// TwinCAT 3 PLC project LabController
// ProgramVersion: 3.1.4022.1
// libraries:
//   Tc2_MC2, * (Beckhoff Automation GmbH)
//   Tc2_Standard, * (Beckhoff Automation GmbH)
//   Tc2_System, * (Beckhoff Automation GmbH)
//   Tc2_Utilities, * (Beckhoff Automation GmbH)
//   Tc3_Module, * (Beckhoff Automation GmbH)
// project tree:
//   DUTs/Control/ ST_Control.TcDUT, ST_ControlComau.TcDUT, ST_ControlStewart.TcDUT, ST_ControlWinch.TcDUT
//   DUTs/ E_MotionLabState.TcDUT
//   DUTs/Feedback/ ST_Feedback.TcDUT, ST_FeedbackComau.TcDUT, ST_FeedbackLeica.TcDUT, ST_FeedbackMru.TcDUT, ST_FeedbackQualisys.TcDUT, ST_FeedbackStewart.TcDUT, ST_FeedbackWinch.TcDUT
//   DUTs/QualisysRT/Components/ ST_3DMarkerPositionNoLabel.TcDUT, ST_3DMarkerPositionNoLabelComponent.TcDUT, ST_RT6D.TcDUT, ST_RT6DComponent.TcDUT
//   DUTs/QualisysRT/ E_ComponentType.TcDUT, ST_RTComponentData.TcDUT, ST_RTDataQRTPacket.TcDUT
//   DUTs/RxHmi/ ST_RxHmi.TcDUT
//   DUTs/RxUdp/ ST_RxUdpComau.TcDUT, ST_RxUdpMru.TcDUT, ST_RxUdpQualisys.TcDUT, ST_RxUdpRemote.TcDUT, ST_RxUdpStewart.TcDUT
//   DUTs/TxHmi/ ST_TxHmi.TcDUT, ST_TxHmiComau.TcDUT, ST_TxHmiMru.TcDUT, ST_TxHmiQualisys.TcDUT, ST_TxHmiStewart.TcDUT, ST_TxHmiWinch.TcDUT
//   DUTs/TxUdp/ ST_TxUdpComau.TcDUT, ST_TxUdpRemote.TcDUT, ST_TxUdpStewart.TcDUT
//   / GVL.TcGVL, MainTask.TcTTO
//   HydroSimulator/ E_TcMatSimDataAreaType.TcDUT, FB_HydroSimulator.TcPOU, FB_TcMatSimObject.TcPOU, ST_HydroSimulatorInitData.TcDUT, ST_HydroSimulator_Input.TcDUT, ST_HydroSimulator_Output.TcDUT, ST_TcMatSimObjectDataAreaInfo.TcDUT
//   POUs/CSV/ FB_CsvReader.TcPOU
//   POUs/Interfaces/ E_ComauMode.TcDUT, E_StewartCommand.TcDUT, E_StewartMode.TcDUT, E_StewartOpMode.TcDUT, E_StewartState.TcDUT, E_StewartStatus.TcDUT, E_WinchMode.TcDUT, FB_ComauInterface.TcPOU, FB_LeicaInterface.TcPOU, FB_MruInterface.TcPOU, FB_QualisysInterface.TcPOU, FB_RemoteInterface.TcPOU, FB_WinchInterface.TcPOU, FB_StewartInterface.TcPOU
//   POUs/ MAIN.TcPOU
//   POUs/Simulink/ FB_QuatToRotMatrix.TcPOU
//   POUs/UdpFBs/ FB_UdpServerRT.TcPOU, FB_UdpClientRT.TcPOU
//   POUs/Utils/ FB_SoftMotion.TcPOU, F_VelocityBoundary.TcPOU, ST_VelocityBoundary.TcDUT
//   SystemFunctions/ CheckDivReal.TcPOU, CheckDivLReal.TcPOU
// real-time tasks:
//   TASK SimTask: cycle T#5ms, priority 21, ADS port 351
//   TASK MainTask: cycle T#5ms, priority 20, ADS port 350
// motion (NC):
//   TASK NC-Task 1 SAF: cycle T#1ms, priority 4, ADS port 501
//   TASK NC-Task 1 SVB: cycle T#5ms, priority 8, ADS port 511
//   AXIS RobotWinch (id 1) // Winch placed on top of Comau Robot
//     General: UnitName=m
//     Dynamic: AccelerationMaximum=10000, DecelerationMaximum=10000, Acceleration=3.56741726765625, Deceleration=3.56741726765625, Jerk=10.7022518029688
//     Velo: RefSearch=0.023782781784375, RefSync=0.023782781784375, SlowManual=0.118913908921875, FastManual=0.71348345353125, Fast=2.3782781784375, Maximum=2.3782781784375
//     OtherSettings: AllowMotionCmdToSlave=true
//     encoder EncType=8
//       EncPara: ScaleFactorNumerator=0.0218304, ScaleFactorDenominator=1048576, Inverse=true, MaxCount=#xffffffff
//         SoftEndMinControl: Enable=true, Range=-7.5
//         SoftEndMaxControl: Enable=true, Range=-6
//     drive DrvType=9
//       DrvPara: Inverse=true, MaxCount=#xffffffff, DriveControlDWord=#x00030100
//         Analog: VeloReferenz=2.61610599628125, VeloScale=1.02400649589962, ScaleFactorActTorque=0.1
//         TimeComp: TaskDelayCycles=1
//     controller CtrType=1
//       CtrPara: PriorControlFactor=1
//         PosDiffControl: Enable=false, Range=10
//         Observer: BandWidth=20
// I/O:
//   DEVICE EM8000 (RT-Ethernet Adapter)
//   DEVICE EM1500 (RT-Ethernet Adapter)
//   DEVICE MRU1 (RT-Ethernet Adapter)
//   DEVICE MRU2 (RT-Ethernet Adapter)
//   DEVICE COMAU (RT-Ethernet Adapter)
//   DEVICE EtherCAT, AmsNetId 169.254.76.98.11.1
//     Drive 1 (AX5103-0000-0210) [AX5103-0000-0210 EtherCAT Drive (SoE, 1 Ch.)]
//     Box 1 (Leica-RT-Output) [Leica RT Output] (disabled)
//   DEVICE REMOTE (RT-Ethernet Adapter)
//   DEVICE QTM (RT-Ethernet Adapter)
// variable links:
//   NC-Task 1 SAF/Axes/RobotWinch <-> EtherCAT/Drive 1 (AX5103-0000-0210)
//     Drive/Inputs/In/nDataIn1 <-> AT/Following distance
//     Drive/Inputs/In/nDcOutputTime <-> InfoData/DcOutputShift
//     Drive/Inputs/In/nState1 <-> AT/Drive status word @bit 8
//     Drive/Inputs/In/nState2 <-> AT/Drive status word
//     Drive/Inputs/In/nState4 @bit 1 <-> WcState/InputToggle
//     Drive/Inputs/In/nState4 <-> WcState/WcState
//     Drive/Outputs/Out/nCtrl1 <-> MDT/Master control word @bit 8
//     Drive/Outputs/Out/nDataOut1 <-> MDT/Position command value
//     Enc/Inputs/In/nDataIn1 <-> AT/Position feedback 1 value
//     Enc/Inputs/In/nDcInputTime <-> InfoData/DcInputShift
//     Enc/Inputs/In/nState4 @bit 1 <-> WcState/InputToggle
//     Enc/Inputs/In/nState4 <-> WcState/WcState
//   LabController/LabController Instance <-> NC-Task 1 SAF/Axes/RobotWinch
//     MainTask Inputs/MAIN.winch.axis.NcToPlc <-> Outputs/ToPlc
//     MainTask Outputs/MAIN.winch.axis.PlcToNc <-> Inputs/FromPlc

CONFIGURATION LabController
    RESOURCE PLC ON TwinCAT3
        TASK MainTask(INTERVAL := T#5ms, PRIORITY := 20);
        PROGRAM MAIN WITH MainTask : MAIN;
    END_RESOURCE
END_CONFIGURATION

// ---- DUTs/Control/ST_Control.TcDUT
TYPE ST_Control :
STRUCT
	em8000: ST_ControlStewart;
	em1500: ST_ControlStewart;
	comau: ST_ControlComau;
	winch: ST_ControlWinch;
END_STRUCT
END_TYPE

// ---- DUTs/Control/ST_ControlComau.TcDUT
TYPE ST_ControlComau :
STRUCT
	u : ARRAY[0..5] OF LREAL;

END_STRUCT
END_TYPE

// ---- DUTs/Control/ST_ControlStewart.TcDUT
TYPE ST_ControlStewart :
STRUCT
	// Velocity setpint to stewart
	u : ARRAY[0..5] OF LREAL;
	
END_STRUCT
END_TYPE

// ---- DUTs/Control/ST_ControlWinch.TcDUT
TYPE ST_ControlWinch :
STRUCT
	length : LREAL;
	length_t : LREAL;
	length_tt : LREAL;
END_STRUCT
END_TYPE

// ---- DUTs/E_MotionLabState.TcDUT
{attribute 'qualified_only'}
{attribute 'strict'}
TYPE E_MotionLabState :
(
	STOP := 16#00,
	NORMAL := 16#01,
	ERROR := 16#10
) USINT;
END_TYPE

// ---- DUTs/Feedback/ST_Feedback.TcDUT
TYPE ST_Feedback :
STRUCT
	em8000: ST_FeedbackStewart;
	em1500: ST_FeedbackStewart;
	mru1: ST_FeedbackMru;
	mru2: ST_FeedbackMru;
	comau: ST_FeedbackComau;
	winch: ST_FeedbackWinch;
	qtm: ST_FeedbackQualisys;
	at960: ST_FeedbackLeica;
END_STRUCT
END_TYPE

// ---- DUTs/Feedback/ST_FeedbackComau.TcDUT
TYPE ST_FeedbackComau :
STRUCT
	q: ARRAY[0..5] OF LREAL;
	q_t: ARRAY[0..5] OF LREAL;
END_STRUCT
END_TYPE

// ---- DUTs/Feedback/ST_FeedbackLeica.TcDUT
TYPE ST_FeedbackLeica :
STRUCT
	pos: ARRAY[0..2] OF LREAL;
	R11: LREAL;
	R12: LREAL;
	R13: LREAL;
	R21: LREAL;
	R22: LREAL;
	R23: LREAL;
	R31: LREAL;
	R32: LREAL;
	R33: LREAL;
END_STRUCT
END_TYPE

// ---- DUTs/Feedback/ST_FeedbackMru.TcDUT
TYPE ST_FeedbackMru :
STRUCT
	eta: ARRAY[0..5] OF LREAL;
	v: ARRAY[0..5] OF LREAL;
END_STRUCT
END_TYPE

// ---- DUTs/Feedback/ST_FeedbackQualisys.TcDUT
TYPE ST_FeedbackQualisys :
STRUCT
	dist: LREAL;
	pos: ARRAY[0..2] OF LREAL;
END_STRUCT
END_TYPE

// ---- DUTs/Feedback/ST_FeedbackStewart.TcDUT
TYPE ST_FeedbackStewart :
STRUCT
	eta: ARRAY[0..5] OF LREAL;
	eta_t: ARRAY[0..5] OF LREAL;
	eta_tt: ARRAY[0..5] OF LREAL;
END_STRUCT
END_TYPE

// ---- DUTs/Feedback/ST_FeedbackWinch.TcDUT
TYPE ST_FeedbackWinch :
STRUCT
	length: LREAL;
	length_t: LREAL;
END_STRUCT
END_TYPE

// ---- DUTs/QualisysRT/Components/ST_3DMarkerPositionNoLabel.TcDUT
TYPE ST_3DMarkerPositionNoLabel :
STRUCT
	x : REAL;
	y : REAL;
	z : REAL;
	id : DINT;
END_STRUCT
END_TYPE

// ---- DUTs/QualisysRT/Components/ST_3DMarkerPositionNoLabelComponent.TcDUT
TYPE ST_3DMarkerPositionNoLabelComponent :
STRUCT
	nSize : UDINT;
	nType : UDINT;
	nMarkers : UDINT;
	nDropRate : INT;
	nOutOfSyncRate : INT;
	markers : ARRAY [0..99] OF ST_3DMarkerPositionNoLabel;
END_STRUCT
END_TYPE

// ---- DUTs/QualisysRT/Components/ST_RT6D.TcDUT
TYPE ST_RT6D :
STRUCT
	x : REAL;
	y : REAL;
	z : REAL;
	rotMatrix : ARRAY [0..8] OF REAL;
END_STRUCT
END_TYPE

// ---- DUTs/QualisysRT/Components/ST_RT6DComponent.TcDUT
TYPE ST_RT6DComponent :
STRUCT
	nSize : UDINT;
	nType : UDINT;
	nBodies : UDINT;
	nDropRate : INT;
	nOutOfSyncRate : INT;
	bodies : ARRAY [0..99] OF ST_RT6D;
END_STRUCT
END_TYPE

// ---- DUTs/QualisysRT/E_ComponentType.TcDUT
{attribute 'qualified_only'}
{attribute 'strict'}
TYPE E_ComponentType :
(
	e3D := 1, // 3D marker data
	e3DNoLabel := 2, //Unidentified 3D marker data
	eAnalog := 3, // Analog data from available analog devices
	eForce := 4, // Force data from available force plates.
	e6D := 5, // 6D data - position and rotation matrix
	e6DEuler := 6, // 6D data - position and Euler angles
	e2D := 7, // 2D marker data
	e2DLinearized := 8, // Linearized 2D marker data
	e3DResiduals := 9, // 3D marker data with residuals
 	e3DNoLabelsResiduals := 10, // Unidentified 3D marker data with residuals
	e6DResiduals := 11, // 6D data - position and rotation matrix with residuals
	e6DEulerResiduals := 12, // 6D data - position and Euler angles with residuals
	eAnalogSingle := 13, // Analog data from available analog devices. Only one sample per channel and camera frame. The latest sample is used if more than one sample is available.
	eImage := 14, // Image frame from a specific camera. Image size and format is set with the XML settings, see Image settings.
	eForceSingle := 15 // Force data from available force plates. Only one sample per plate and camera frame. The latest sample is used if more than one sample is available.
);
END_TYPE

// ---- DUTs/QualisysRT/ST_RTComponentData.TcDUT
TYPE ST_RTComponentData :
STRUCT
	nSize : UDINT;
	nType : UDINT;
END_STRUCT
END_TYPE

// ---- DUTs/QualisysRT/ST_RTDataQRTPacket.TcDUT
TYPE ST_RTDataQRTPacket :
STRUCT
	nSize : UDINT;
	nType : UDINT;
	nTimestamp : LINT;
	nFramenumber : UDINT;
	nComponentCount : UDINT;
END_STRUCT
END_TYPE

// ---- DUTs/RxHmi/ST_RxHmi.TcDUT
TYPE ST_RxHmi :
STRUCT
	counter : UDINT := 0;
	winchJogUp : BOOL;
	winchJogDown : BOOL;
	xboxLeftX : REAL;
	xboxLeftY : REAL;
	xboxRightX : REAL;
	xboxRightY : REAL;
	xboxLT : REAL;
	xboxRT : REAL;
END_STRUCT
END_TYPE

// ---- DUTs/RxUdp/ST_RxUdpComau.TcDUT
TYPE ST_RxUdpComau :
STRUCT
	frameCounter : DINT := 0;
	q 		: ARRAY [0..5] OF REAL;
	q_t 	: ARRAY [0..5] OF REAL;
	qMin 	: ARRAY [0..5] OF REAL;
	qMax 	: ARRAY [0..5] OF REAL;
	qMax_t 	: ARRAY [0..5] OF REAL;
END_STRUCT
END_TYPE

// ---- DUTs/RxUdp/ST_RxUdpMru.TcDUT
{attribute 'pack_mode' := '1'}
TYPE ST_RxUdpMru :
STRUCT
	mruOK : BYTE; // Mru Status, 113=OK
	dataLength : BYTE; // Data length
	token : BYTE; // MRU token
	SystemTime : DINT; // No. 176 - [ms] - Sample time in milliseconds since power on
	SensorTemp : REAL; // No. 31 - [DegC] - Sensor house temprature     
	AngRate_D : REAL; // No. 9 - [rad/s] - Angular rate in Down direction (h-frame). Turn Rate
	Roll : REAL; // No. 63 - [rad] - Roll angle (euler angle)
	Pitch : REAL; // No. 64 - [rad] - Pitch angle (euler angle)
	Yaw : REAL; // No. 65 - [rad] - Yaw angle (euler angle)
	AngRate_R : REAL; // No. 1 - [rad/s] - Angular rate in roll axis (b-frame)
	AngRate_P : REAL; // No. 2 - [rad/s] - Angular rate in pitch axis (b-frame)
	AngRate_Y : REAL; // No. 3 - [rad/s] - Angular rate in yaw axis (b-frame)
	VelMru_R : REAL; // No. 244 - [m/s] - Linear velocity at MRU point in R-direction (b-frame)
	VelMru_P : REAL; // No. 245 - [m/s] - Linear velocity at MRU point in P-direction (b-frame)
	VelMru_Y : REAL; // No. 246 - [m/s] - Linear velocity at MRU point in Y-direction (b-frame)
	AccMru_R : REAL; // No. 238 - [m/s] - Linear acceleration at MRU point in R-direction (b-frame)
	AccMru_P : REAL; // No. 239 - [m/s] - Linear acceleration at MRU point in P-direction (b-frame)
	AccMru_Y : REAL; // No. 240 - [m/s] - Linear acceleration at MRU point in Y-direction (b-frame)
	PosCg_F : REAL; // No. 274 - [m] - Linear position at CG in forward direction (h-frame)
	PosCg_S : REAL; // No. 275 - [m] - Linear position at CG in starboard direction (h-frame)
	PosCg_D : REAL; // No. 276 - [m] - Linear position at CG in down direction (h-frame)
	VelCg_F : REAL; // No. 262 - [m/s] - Linear velocity at CG in forward direction (h-frame)
	VelCg_S : REAL; // No. 263 - [m/s] - Linear velocity at CG in starboard direction (h-frame)
	VelCg_D : REAL; // No. 264 - [m/s] - Linear velocity at CG in down direction (h-frame)
	AccCg_F : REAL; // No. 250 - [m/s2] - Linear acceleration (raw/unfiltered) at CG in forward direction (h-frame)
	AccCg_S : REAL; // No. 251 - [m/s2] - Linear acceleration (raw/unfiltered) at CG in starboard direction (h-frame)
	AccCg_D : REAL; // No. 252 - [m/s2] - Linear acceleration (raw/unfiltered) at CG in down direction (h-frame)
	checksum : BYTE; // Data checksum 
END_STRUCT
END_TYPE

// ---- DUTs/RxUdp/ST_RxUdpQualisys.TcDUT
TYPE ST_RxUdpQualisys :
STRUCT
	// Header
	dataSize : UDINT;
	dataType : UDINT;
	timestamp : ULINT;
	frameNumber : UDINT;
	componentCount : UDINT;
	// Component
	componentSize : UDINT;
	componentType : UDINT;
END_STRUCT
END_TYPE

// ---- DUTs/RxUdp/ST_RxUdpRemote.TcDUT
TYPE ST_RxUdpRemote :
STRUCT
	iUdpKey : UDINT; // Udp Key
	iCounter : UDINT; // Heartbeat counter
	eModeCmd : UDINT; // Operation mode
	em8000_u : ARRAY [0..5] OF REAL; // EM8000 DOF position setpoints
	em8000_u_t : ARRAY [0..5] OF REAL; // EM8000 DOF velocity setpoints
	em1500_u : ARRAY [0..5] OF REAL; // EM1500 DOF position setpoints
	em1500_u_t : ARRAY [0..5] OF REAL; // EM1500 DOF velocity setpoints
	comau_u : ARRAY [0..5] OF REAL; // Joint speed setpoints
	winch_u : REAL; // Winch wire speed setpoint
	
END_STRUCT
END_TYPE

// ---- DUTs/RxUdp/ST_RxUdpStewart.TcDUT
TYPE ST_RxUdpStewart :
STRUCT
	Frame_Count : UDINT := 0;
	Motion_Status : UDINT := 0;
	Platform_setpoint_surge : REAL := 0.0;
	Platform_setpoint_sway : REAL := 0.0;
	Platform_setpoint_heave : REAL := 0.0;
	Platform_setpoint_roll : REAL := 0.0;
	Platform_setpoint_pitch : REAL := 0.0;
	Platform_setpoint_yaw : REAL := 0.0;
	Special_effect_surge_setpoint : REAL := 0.0;
	Special_effect_sway_setpoint : REAL := 0.0;
	Special_effect_heave_setpoint : REAL := 0.0;
	Special_effect_roll_setpoint : REAL := 0.0;
	Special_effect_pitch_setpoint : REAL := 0.0;
	Special_effect_yaw_setpoint : REAL := 0.0;
	Actual_position_actuator_1 : REAL := 0.0;
	Actual_position_actuator_2 : REAL := 0.0;
	Actual_position_actuator_3 : REAL := 0.0;
	Actual_position_actuator_4 : REAL := 0.0;
	Actual_position_actuator_5 : REAL := 0.0;
	Actual_position_actuator_6 : REAL := 0.0;
	Actual_platform_position_surge : REAL := 0.0;
	Actual_platform_position_sway : REAL := 0.0;
	Actual_platform_position_heave : REAL := 0.0;
	Actual_platform_position_roll : REAL := 0.0;
	Actual_platform_position_pitch : REAL := 0.0;
	Actual_platform_position_yaw : REAL := 0.0;
	Actual_platform_velocity_surge : REAL := 0.0;
	Actual_platform_velocity_sway : REAL := 0.0;
	Actual_platform_velocity_heave : REAL := 0.0;
	Actual_platform_velocity_roll : REAL := 0.0;
	Actual_platform_velocity_pitch : REAL := 0.0;
	Actual_platform_velocity_yaw : REAL := 0.0;
	Actual_platform_acceleration_surge : REAL := 0.0;
	Actual_platform_acceleration_sway : REAL := 0.0;
	Actual_platform_acceleration_heave : REAL := 0.0;
	Actual_platform_acceleration_roll : REAL := 0.0;
	Actual_platform_acceleration_pitch : REAL := 0.0;
	Actual_platform_acceleration_yaw : REAL := 0.0;
END_STRUCT
END_TYPE

// ---- DUTs/TxHmi/ST_TxHmi.TcDUT
TYPE ST_TxHmi :
STRUCT
	em8000 : ST_TxHmiStewart;
	em1500 : ST_TxHmiStewart;
	mru1 : ST_TxHmiMru;
	mru2 : ST_TxHmiMru;
	comau : ST_TxHmiComau;
	winch : ST_TxHmiWinch;
	qtm : ST_TxHmiQualisys;
	phi : ARRAY [0..1] OF REAL;
	phi_t : ARRAY [0..1] OF REAL;	
	e : ARRAY [0..2] OF REAL;
	c : REAL;
END_STRUCT
END_TYPE

// ---- DUTs/TxHmi/ST_TxHmiComau.TcDUT
TYPE ST_TxHmiComau :
STRUCT
	status : DINT;
	u : ARRAY [0..5] OF REAL;
	q : ARRAY [0..5] OF REAL;
	q_t : ARRAY [0..5] OF REAL;
	qMin : ARRAY [0..5] OF REAL;
	qMax : ARRAY [0..5] OF REAL;
	qMax_t : ARRAY [0..5] OF REAL;
END_STRUCT
END_TYPE

// ---- DUTs/TxHmi/ST_TxHmiMru.TcDUT
TYPE ST_TxHmiMru :
STRUCT
	status : DINT := 0;
	eta : ARRAY [0..5] OF REAL;
END_STRUCT
END_TYPE

// ---- DUTs/TxHmi/ST_TxHmiQualisys.TcDUT
TYPE ST_TxHmiQualisys :
STRUCT
	status : DINT;
	dist : REAL;
	x : REAL;
	y : REAL;
	z : REAL;
	markers : ARRAY [0..9] OF ST_3DMarkerPositionNoLabel;
END_STRUCT
END_TYPE

// ---- DUTs/TxHmi/ST_TxHmiStewart.TcDUT
TYPE ST_TxHmiStewart :
STRUCT
	status : DINT := 0;
	eta : ARRAY [0..5] OF REAL;
	etaRef : ARRAY [0..5] OF REAL;
	cyl : ARRAY [0..5] OF REAL;
	dofScale : ARRAY [0..5] OF REAL;
END_STRUCT
END_TYPE

// ---- DUTs/TxHmi/ST_TxHmiWinch.TcDUT
TYPE ST_TxHmiWinch :
STRUCT
	status : DINT := 0;
	l : REAL;
END_STRUCT
END_TYPE

// ---- DUTs/TxUdp/ST_TxUdpComau.TcDUT
TYPE ST_TxUdpComau :
STRUCT
	udpKey : DINT := 0;
	cmnd : DINT; // 0: SETTLED, 1: ENGAGED
	qDotRef : ARRAY [0..5] OF REAL;
END_STRUCT
END_TYPE

// ---- DUTs/TxUdp/ST_TxUdpRemote.TcDUT
TYPE ST_TxUdpRemote :
STRUCT
	// Mode and time
	eMode : UDINT;
	t : REAL;
	
	// Equipement: Comau robot
	comau_q : ARRAY [0..5] OF REAL;
	comau_q_t : ARRAY [0..5] OF REAL;
	
	// Equipement: Robot Winch
	winch_l : REAL;
	winch_l_t : REAL;

	// Equipement: EM8000
	em8000_eta : ARRAY [0..5] OF REAL;
	em8000_eta_t : ARRAY [0..5] OF REAL;
	em8000_eta_tt : ARRAY [0..5] OF REAL;
	
	// Equipement: MRU1 (Mounted on EM8000)
	mru1_eta : ARRAY [0..5] OF REAL;
	mru1_v : ARRAY [0..5] OF REAL;
	
	// Equipement: EM1500 and MRU2
	em1500_eta : ARRAY [0..5] OF REAL;
	em1500_eta_t : ARRAY [0..5] OF REAL;
	em1500_eta_tt : ARRAY [0..5] OF REAL;
	
	// Equipement: MRU2 (Mounted on EM1500)
	mru2_eta : ARRAY [0..5] OF REAL;
	mru2_v : ARRAY [0..5] OF REAL;
	
END_STRUCT
END_TYPE

// ---- DUTs/TxUdp/ST_TxUdpStewart.TcDUT
TYPE ST_TxUdpStewart :
STRUCT
	COUNT : UDINT := 0;
	CMND : UDINT := 0;
	AX : REAL := 0.0;
	AY : REAL := 0.0;
	AZ : REAL := 0.0;
	Dax : REAL := 0.0;
	Day : REAL := 0.0;
	Daz : REAL := 0.0;
	P_dot_CG : REAL := 0.0;
	Q_dot_CG : REAL := 0.0;
	R_dot_CG : REAL := 0.0;
	P_CG : REAL := 0.0;
	Q_CG : REAL := 0.0;
	R_CG : REAL := 0.0;
	Phi : REAL := 0.0;
	Theta : REAL := 0.0;
	U : REAL := 0.0;
	X_DIRECT : REAL := 0.0;
	Y_DIRECT : REAL := 0.0;
	Z_DIRECT : REAL := 0.0;
	X_CG : REAL := 0.0;
	Y_CG : REAL := 0.0;
	Z_CG : REAL := 0.0;
	Flags : REAL := 0.0;
	Bump_1 : REAL := 0.0;
	Bump_2 : REAL := 0.0;
	Bump_3 : REAL := 0.0;
	Bump_4 : REAL := 0.0;
	Bump_5 : REAL := 0.0;
	FREQ1 : REAL := 0.0;
	FREQ2 : REAL := 0.0;
	FREQ3 : REAL := 0.0;
	FREQ4 : REAL := 0.0;
	FREQ5 : REAL := 0.0;
	FREQ6 : REAL := 0.0;
	FREQ7 : REAL := 0.0;
	FREQ8 : REAL := 0.0;
	FREQ9 : REAL := 0.0;
	FREQ10 : REAL := 0.0;
	FREQ11 : REAL := 0.0;
	FREQ12 : REAL := 0.0;
	FREQ13 : REAL := 0.0;
	FREQ14 : REAL := 0.0;
	FREQ15 : REAL := 0.0;
	FREQ16 : REAL := 0.0;
	FREQ17 : REAL := 0.0;
	FREQ18 : REAL := 0.0;
	FREQ19 : REAL := 0.0;
	FREQ20 : REAL := 0.0;
	XGAIN1 : REAL := 0.0;
	XGAIN2 : REAL := 0.0;
	XGAIN3 : REAL := 0.0;
	XGAIN4 : REAL := 0.0;
	XGAIN5 : REAL := 0.0;
	XGAIN6 : REAL := 0.0;
	XGAIN7 : REAL := 0.0;
	XGAIN8 : REAL := 0.0;
	XGAIN9 : REAL := 0.0;
	XGAIN10 : REAL := 0.0;
	XGAIN11 : REAL := 0.0;
	XGAIN12 : REAL := 0.0;
	XGAIN13 : REAL := 0.0;
	XGAIN14 : REAL := 0.0;
	XGAIN15 : REAL := 0.0;
	XGAIN16 : REAL := 0.0;
	XGAIN17 : REAL := 0.0;
	XGAIN18 : REAL := 0.0;
	XGAIN19 : REAL := 0.0;
	XGAIN20 : REAL := 0.0;
	YGAIN1 : REAL := 0.0;
	YGAIN2 : REAL := 0.0;
	YGAIN3 : REAL := 0.0;
	YGAIN4 : REAL := 0.0;
	YGAIN5 : REAL := 0.0;
	YGAIN6 : REAL := 0.0;
	YGAIN7 : REAL := 0.0;
	YGAIN8 : REAL := 0.0;
	YGAIN9 : REAL := 0.0;
	YGAIN10 : REAL := 0.0;
	YGAIN11 : REAL := 0.0;
	YGAIN12 : REAL := 0.0;
	YGAIN13 : REAL := 0.0;
	YGAIN14 : REAL := 0.0;
	YGAIN15 : REAL := 0.0;
	YGAIN16 : REAL := 0.0;
	YGAIN17 : REAL := 0.0;
	YGAIN18 : REAL := 0.0;
	YGAIN19 : REAL := 0.0;
	YGAIN20 : REAL := 0.0;
	ZGAIN1 : REAL := 0.0;
	ZGAIN2 : REAL := 0.0;
	ZGAIN3 : REAL := 0.0;
	ZGAIN4 : REAL := 0.0;
	ZGAIN5 : REAL := 0.0;
	ZGAIN6 : REAL := 0.0;
	ZGAIN7 : REAL := 0.0;
	ZGAIN8 : REAL := 0.0;
	ZGAIN9 : REAL := 0.0;
	ZGAIN10 : REAL := 0.0;
	ZGAIN11 : REAL := 0.0;
	ZGAIN12 : REAL := 0.0;
	ZGAIN13 : REAL := 0.0;
	ZGAIN14 : REAL := 0.0;
	ZGAIN15 : REAL := 0.0;
	ZGAIN16 : REAL := 0.0;
	ZGAIN17 : REAL := 0.0;
	ZGAIN18 : REAL := 0.0;
	ZGAIN19 : REAL := 0.0;
	ZGAIN20 : REAL := 0.0;
	X_EXTRA : REAL := 0.0;
	Y_EXTRA : REAL := 0.0;
	Z_EXTRA : REAL := 0.0;
	PHI_EXTRA : REAL := 0.0;
	THETA_EXTRA : REAL := 0.0;
	PSI_EXTRA : REAL := 0.0;
	X_EXTRA_DOT : REAL := 0.0;
	Y_EXTRA_DOT : REAL := 0.0;
	Z_EXTRA_DOT : REAL := 0.0;
	PHI_EXTRA_DOT : REAL := 0.0;
	THETA_EXTRA_DOT : REAL := 0.0;
	PSI_EXTRA_DOT : REAL := 0.0;
	X_EXTRA_DDOT : REAL := 0.0;
	Y_EXTRA_DDOT : REAL := 0.0;
	Z_EXTRA_DDOT : REAL := 0.0;
	PHI_EXTRA_DDOT : REAL := 0.0;
	THETA_EXTRA_DDOT : REAL := 0.0;
	PSI_EXTRA_DDOT : REAL := 0.0;
END_STRUCT
END_TYPE

// ---- HydroSimulator/E_TcMatSimDataAreaType.TcDUT
TYPE E_TcMatSimDataAreaType :
(
	NotSpecified := 0,
	Standard,
	InputSrc,
	InputDst,
	OutputSrc,
	OutputDst,
	InternalDa,
	MArea,
	RetainDa
);
END_TYPE

// ---- HydroSimulator/ST_HydroSimulatorInitData.TcDUT
{attribute 'pack_mode' := '4'}
TYPE ST_HydroSimulatorInitData :
STRUCT
	Header: TComInitDataHdr;
	CallByHdr: TComInitDataElmHdr;
	CallBy: TctModuleCallByType;
	ExecutionSequenceHdr: TComInitDataElmHdr;
	ExecutionSequence: TctModuleExecutionSequenceType;
	StepSizeHdr: TComInitDataElmHdr;
	StepSize: TctStepSizeType;
	ExecuteModelCodeHdr: TComInitDataElmHdr;
	ExecuteModelCode: BOOL;
	ModelParametersHdr: TComInitDataElmHdr;
	ModelParameters: P_HydroSimulator_T;
	ContextInfoArr_0_TaskOidHdr: TComInitDataElmHdr;
	ContextInfoArr_0_TaskOid: OTCID;
	ContextInfoArr_0_TaskPriorityHdr: TComInitDataElmHdr;
	ContextInfoArr_0_TaskPriority: UDINT;
	ContextInfoArr_0_TaskCycleTimeNsHdr: TComInitDataElmHdr;
	ContextInfoArr_0_TaskCycleTimeNs: UDINT;
	ContextInfoArr_0_TaskPortHdr: TComInitDataElmHdr;
	ContextInfoArr_0_TaskPort: UINT;
	ContextInfoArr_0_TaskSortOrderHdr: TComInitDataElmHdr;
	ContextInfoArr_0_TaskSortOrder: UDINT;
END_STRUCT
END_TYPE

// ---- HydroSimulator/ST_HydroSimulator_Input.TcDUT
TYPE ST_HydroSimulator_Input :
STRUCT
	bReset: BOOL;
	etaMax: matrix_6_real_T := [0.1, 0.1, 0.3, 5.0/180.0*PI, 5.0/180.0*PI, 5.0/180.0*PI];
	w0 : LREAL := 0.5457;
	lambda : LREAL := 0.2405;
	sigma : LREAL := 0.8444;
	
END_STRUCT
END_TYPE

// ---- HydroSimulator/ST_HydroSimulator_Output.TcDUT
TYPE ST_HydroSimulator_Output :
STRUCT
	scale: matrix_6_real_T;
	eta: matrix_6_real_T;
	v: matrix_6_real_T;
	v_t: matrix_6_real_T;
END_STRUCT
END_TYPE

// ---- HydroSimulator/ST_TcMatSimObjectDataAreaInfo.TcDUT
TYPE ST_TcMatSimObjectDataAreaInfo :
STRUCT
	pPlcVar: PVOID;
	pModuleProcImg: PVOID;
	nSize: UDINT;
	nDataAreaId: UDINT;
	eDataAreaType: E_TcMatSimDataAreaType;
END_STRUCT
END_TYPE

// ---- POUs/Interfaces/E_ComauMode.TcDUT
{attribute 'qualified_only'}
{attribute 'strict'}
TYPE E_ComauMode :
(
	SETTLED := 0,
	REMOTE,
	MOTION_COMP
) DINT;
END_TYPE

// ---- POUs/Interfaces/E_StewartCommand.TcDUT
{attribute 'qualified_only'}
{attribute 'strict'}
TYPE E_StewartCommand :
(
	TO_OFF	 		:= 16#00000000,
	TO_SETTLED 		:= 16#00000001,
	TO_NEUTRAL 		:= 16#00000003,
	TO_ENGAGED 		:= 16#00000007,
	ACK_FAULT 		:= 16#00000011 // Akcnowledge fault and go to settled
) UDINT;
END_TYPE

// ---- POUs/Interfaces/E_StewartMode.TcDUT
{attribute 'qualified_only'}
{attribute 'strict'}
TYPE E_StewartMode :
(
	SETTLED := 0,
	NEUTRAL,
	SIMULATION,
	GENERATOR,
	REMOTE
) USINT ;
END_TYPE

// ---- POUs/Interfaces/E_StewartOpMode.TcDUT
{attribute 'qualified_only'}
{attribute 'strict'}
TYPE E_StewartOpMode :
(
	MANUAL 	:= 16#00,
	NORMAL	:= 16#01
) USINT;
END_TYPE

// ---- POUs/Interfaces/E_StewartState.TcDUT
{attribute 'qualified_only'}
{attribute 'strict'}
TYPE E_StewartState :
(
	TRANSIT 		:= 16#00,
	OFF				:= 16#01,
	SETTLED			:= 16#02,
	OIL_HEATING		:= 16#03,
	NEUTRAL 		:= 16#04,
	NEUTRAL_FREEZE	:= 16#05,
	ENGAGED			:= 16#08,
	ENGAGED_FREEZE	:= 16#09	
) USINT;
END_TYPE

// ---- POUs/Interfaces/E_StewartStatus.TcDUT
{attribute 'qualified_only'}
{attribute 'strict'}
TYPE E_StewartStatus :
(
	SYSTEM_OK 	:= 16#00,
	WARNING		:= 16#04,
	ERROR		:= 16#08
) USINT;
END_TYPE

// ---- POUs/Interfaces/E_WinchMode.TcDUT
{attribute 'qualified_only'}
{attribute 'strict'}
TYPE E_WinchMode :
(
	SETTLED := 0,
	LOCAL,
	REMOTE,
	MOTION_COMP
) USINT;
END_TYPE

// ---- POUs/Utils/ST_VelocityBoundary.TcDUT
TYPE ST_VelocityBoundary :
STRUCT
	qMin_t : LREAL;
	qMax_t : LREAL;
END_STRUCT
END_TYPE

// ---- GVL.TcGVL
{attribute 'qualified_only'}
VAR_GLOBAL
	logMessage : STRING(255) := 'No Message';
END_VAR

// ---- POUs/MAIN.TcPOU
PROGRAM MAIN
VAR_INPUT
	bStop : BOOL;
	bReset : BOOL := FALSE;
	
END_VAR
VAR_OUTPUT
	eState : E_MotionLabState;
	
END_VAR
VAR
	// TEST/DEBUG
	rand : DRAND;
	k : UINT;
	data : ARRAY [0..9] OF REAL;

	// Task monitoring
	fbGetCurrentTaskIdx : GETCURTASKINDEX;
	bCycleTimeExceeded : BOOL;
	nCycleCount : UDINT;
	Ts : LREAL;
	t : LREAL;
	
	// Linear wave parameters, Hs = 8 and Tp = 12.0;
	w0 AT %Q* : LREAL := 0.5457;
	lambda AT %Q* : LREAL := 0.2405;
	sigma AT %Q* : LREAL := 1.5012;
	
	// HMI data
	txHmi : ST_TxHmi;
	rxHmi : ST_RxHmi;
	
	// HMI activity check
	hmiCounterOld : UDINT := 0;
	hmiTimer : TON;
	
	// Remote interface
	remote : FB_RemoteInterface('192.168.90.60', 50060, 50050); // CPU-X001
	
	// Machinery
	em8000 : FB_StewartInterface('192.168.90.30', 50030, 50040, oid:=16#01010060);
	em1500 : FB_StewartInterface('192.168.90.31', 50031, 50041, oid:=16#01010070);
	comau : FB_ComauInterface('192.168.90.32', 50032, 50042);
	winch : FB_WinchInterface(ADR(txHmi.winch));
	
	// Sensors
	mru1 : FB_MruInterface(50043, ADR(txHmi.mru1));
	mru2 : FB_MruInterface(50044, ADR(txHmi.mru2));
	qtm : FB_QualisysInterface(50199, ADR(txHmi.qtm));
	at960 : FB_LeicaInterface;
	
	// Hydro simulators
	
	
	
	// System call for starting PqQt HMI
	fbStartProcess : NT_StartProcess;
	
	phi : ARRAY [0..1] OF LREAL;
END_VAR

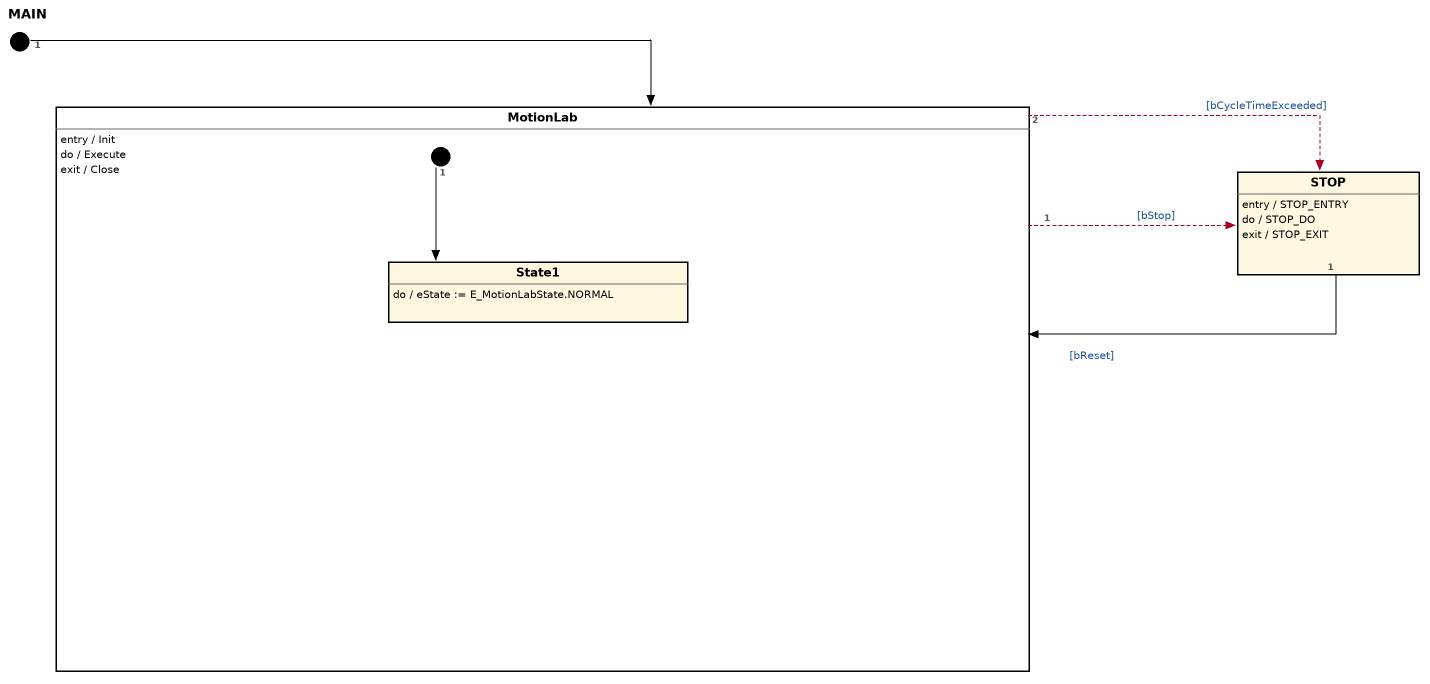
STATECHART MAIN  // abortable
    START StartState1
    COMPOSITE STATE MotionLab
        entry / Init
        do / Execute
        exit / Close
        START StartState2
        STATE State1
            do / eState := E_MotionLabState.NORMAL
        StartState2 -> State1  // priority 1, on completion
    END_STATE
    STATE STOP
        entry / STOP_ENTRY
        do / STOP_DO
        exit / STOP_EXIT
    StartState1 -> MotionLab  // priority 1, on completion
    MotionLab -> STOP [bStop] // priority 1, exception
    MotionLab -> STOP [bCycleTimeExceeded] // priority 2, exception
    STOP -> MotionLab [bReset] // priority 1
END_STATECHART

METHOD Close : BOOL
VAR_INPUT
END_VAR
END_METHOD

METHOD PRIVATE Execute : BOOL
VAR_INPUT
END_VAR
VAR
	i : UINT;

END_VAR
// Task monitoring
fbGetCurrentTaskIdx();
bCycleTimeExceeded := _TaskInfo[fbGetCurrentTaskIdx.index].CycleTimeExceeded;
nCycleCount := _TaskInfo[fbGetCurrentTaskIdx.index].CycleCount;
Ts := UDINT_TO_LREAL(_TaskInfo[fbGetCurrentTaskIdx.index].CycleTime/10)/1E6;


FOR i := 0 TO 9 DO
	data[i] := LREAL_TO_REAL((1 + i)*0.1*SIN(0.1*2*PI*t));
END_FOR

// Update all interfaces
em8000(
	Ts := Ts,
);
em1500(
	Ts := Ts,
);

mru1();
mru2();
at960();
qtm();
comau();

winch(
	Ts := Ts
);


// *** REMOTE Interface ***
// PLC -> REMOTE
remote.feedback.em8000 := em8000.feedback;
remote.feedback.mru1 := mru1.feedback;

remote.feedback.em1500 := em1500.feedback;
remote.feedback.mru2 := mru2.feedback;

remote.feedback.comau.q := comau.q;

// Execute remote
remote(
	Ts := Ts
);

// REMOTE -> PLC
em1500.bRemoteActive := remote.bActive;
em1500.uRemote := remote.control.em1500.u;
em1500.uRemote_t := remote.control.em1500.u_t;

// *** REMOTE Interface ***
END_METHOD

METHOD Init : BOOL
VAR_INPUT
END_VAR
END_METHOD

METHOD PRIVATE STOP_DO : BOOL
VAR_INPUT
END_VAR

// Update all interfaces
Execute();

eState := E_MotionLabState.STOP;
END_METHOD

METHOD PRIVATE STOP_ENTRY : BOOL
VAR_INPUT
END_VAR
em8000.bStop := TRUE;
em1500.bStop := TRUE;
END_METHOD

METHOD PRIVATE STOP_EXIT : BOOL
VAR_INPUT
END_VAR
bStop := FALSE;
bReset := FALSE;

// Reset equipement
em8000.bReset := TRUE;
em1500.bReset := TRUE;
END_METHOD

END_PROGRAM

// ---- POUs/Interfaces/FB_RemoteInterface.TcPOU
FUNCTION_BLOCK FB_RemoteInterface
VAR_INPUT
	Ts : LREAL := 0.005;
	// feedback from motion lab
	feedback : ST_Feedback;
	
	
END_VAR
VAR_OUTPUT
	// Activity status
	bActive : BOOL := FALSE;
	
	// Control to motion lab
	control : ST_Control;
	
END_VAR
VAR
	// Udp connection
	rxUdp : ST_RxUdpRemote;
	txUdp : ST_TxUdpRemote;
	udpClient : FB_UdpClientRT('', 0, 0, 0, 0, 0, 0);	// Dummy constructor
	
	// Timer
	iCounterOld : UDINT := 0;
	fbTimer : TON;
	
	
	i : UINT;
	
END_VAR

// Feedback data
FOR i := 0 TO 5 DO
	// eMode
	txUdp.eMode := 0;
	
	// Time 
	txUdp.t := txUdp.t + LREAL_TO_REAL(Ts);
	
	// EM8000
	txUdp.em8000_eta[i] := LREAL_TO_REAL(feedback.em8000.eta[i]);
	txUdp.em8000_eta_t[i] := LREAL_TO_REAL(feedback.em8000.eta_t[i]);
	txUdp.em8000_eta_tt[i] := LREAL_TO_REAL(feedback.em8000.eta_tt[i]);
	
	// MRU1
	txUdp.mru1_eta[i] := LREAL_TO_REAL(feedback.mru1.eta[i]);
	txUdp.mru1_v[i] := LREAL_TO_REAL(feedback.mru1.v[i]);
	
	// EM1500
	txUdp.em1500_eta[i] := LREAL_TO_REAL(feedback.em1500.eta[i]);
	txUdp.em1500_eta_t[i] := LREAL_TO_REAL(feedback.em1500.eta_t[i]);
	txUdp.em1500_eta_tt[i] := LREAL_TO_REAL(feedback.em1500.eta_tt[i]);
	
	// MRU1
	txUdp.mru2_eta[i] := LREAL_TO_REAL(feedback.mru2.eta[i]);
	txUdp.mru2_v[i] := LREAL_TO_REAL(feedback.mru2.v[i]);
	
	
	// COMAU
	
	
	
END_FOR

// WINCH



// Update Udp client
udpClient();

// Control data
FOR i := 0 TO 5 DO
	// EM8000
	control.em8000.u[i] := REAL_TO_LREAL(rxUdp.em8000_u[i]);
	
	// MRU1
	
	
	// EM1500
	control.em1500.u[i] := REAL_TO_LREAL(rxUdp.em1500_u[i]);
	
	// MRU2
	
	// COMAU
	
	
END_FOR

// WINCH




// Timeout setting
fbTimer.PT := T#500MS;

IF rxUdp.iCounter <> iCounterOld THEN
	// Update old counter
	iCounterOld := rxUdp.iCounter;
	
	// Reset timeout timer
	fbTimer(
		IN := FALSE
	);
	
ELSE
	// Start timout timer
	fbTimer(
		IN := TRUE
	);
	
END_IF

// Set bActive based on timer
bActive := NOT fbTimer.Q;

METHOD FB_exit : BOOL
VAR_INPUT
	bInCopyCode : BOOL; // if TRUE, the exit method is called for exiting an instance that is copied afterwards (online change).
END_VAR
END_METHOD

METHOD FB_init : BOOL
VAR_INPUT
	bInitRetains : BOOL; // if TRUE, the retain variables are initialized (warm start / cold start)
	bInCopyCode : BOOL;  // if TRUE, the instance afterwards gets moved into the copy code (online change)
	
	// Init variables
	_remoteIpAddr : T_Ipv4Addr;
	_remotePort : UINT;
	_localPort : UINT;
END_VAR
// Initilize udpClient
udpClient.FB_init(
	bInitRetains,
	bInCopyCode,
	_remoteIpAddr,
	_remotePort,
	_localPort,
	SIZEOF(rxUdp),
	ADR(rxUdp),
	SIZEOF(txUdp),
	ADR(txUdp)
);
END_METHOD

METHOD FB_reinit : BOOL
VAR_INPUT
END_VAR
END_METHOD

END_FUNCTION_BLOCK

// ---- POUs/UdpFBs/FB_UdpClientRT.TcPOU
{attribute 'c++_compatible'}
FUNCTION_BLOCK FB_UdpClientRT IMPLEMENTS ITcIoUdpProtocolRecv
VAR_INPUT
	
END_VAR
VAR_OUTPUT
END_VAR
VAR
	// ITcIoUdpProtocolRecv related 
	{attribute 'TcInitSymbol'}
	oid : OTCID; 
	ipUdp : ITcIoUdpProtocol;
	
	// Initilized variables
	remoteIpAddr : UDINT;
	remotePort : UINT;
	localPort : UINT;
	{attribute 'tc_no_symbol'}
	nRxData : UDINT := 0;
	{attribute 'tc_no_symbol'}
	pRxData : PVOID;
	{attribute 'tc_no_symbol'}
	nTxData : UDINT := 0;
	{attribute 'tc_no_symbol'}
	pTxData : PVOID;
	
	// Send/Recv counters
	rxCounter : UINT;
	txCounter : UINT;
	
	// Result
	hrInit : HRESULT;
	hrSend : HRESULT;
END_VAR

IF ipUdp <> 0 THEN
	// Send data to remote server
	IF nTxData > 0 THEN		
		hrSend := ipUdp.SendData(remoteIpAddr, remotePort, localPort, nTxData, pTxData, TRUE, 0);
		txCounter := txCounter + 1;
	END_IF
	
	// Check for incoming data
	IF nRxData > 0 THEN
		ipUdp.CheckReceived();
	END_IF
END_IF

{attribute 'conditionalshow'}
METHOD FB_exit : BOOL
VAR_INPUT
	bInCopyCode : BOOL; // if TRUE, the exit method is called for exiting an instance that is copied afterwards (online change).
END_VAR
IF NOT bInCopyCode THEN // no online change
	IF ipUdp <> 0 THEN 
		ipUdp.UnregisterReceiver(localPort); // Shutdown
		FW_SafeRelease(ADR(ipUdp));
		FB_exit := TRUE; 
	END_IF
END_IF
END_METHOD

{attribute 'conditionalshow'}
METHOD FB_init : BOOL
VAR_INPUT
	bInitRetains : BOOL; // if TRUE, the retain variables are initialized (warm start / cold start)
	bInCopyCode : BOOL;  // if TRUE, the instance afterwards gets moved into the copy code (online change)
	
	// Init variables
	_remoteIpAddr : T_Ipv4Addr;
	_remotePort : UINT;
	_localPort : UINT;
	_nRxData : UDINT;
	_pRxData : PVOID;
	_nTxData : UDINT;
	_pTxData : PVOID;
END_VAR
VAR
    ipSrv : ITComObjectServer;
	ipArr : T_IPv4AddrArr;
	i : UINT;
END_VAR
// Initilize member variables
remoteIpAddr := IpToLong(_remoteIpAddr);
remotePort := _remotePort;
localPort := _localPort;
nRxData := _nRxData;
pRxData := _pRxData;
nTxData := _nTxData;
pTxData := _pTxData;

IF NOT bInCopyCode THEN // no online change
	IF ipUdp = 0 THEN
	    hrInit := FW_ObjMgr_GetObjectInstance(
			oid:=oid, 
			iid:=TC_GLOBAL_IID_LIST.IID_ITcIoUdpProtocol, 
			pipUnk:=ADR(ipUdp)
		);
		
		IF SUCCEEDED(hrInit) THEN 
			IF  SUCCEEDED(ipUdp.RegisterReceiver(localPort, THIS^)) THEN //open port
				FB_init := TRUE;
			ELSE 
				FW_SafeRelease(ADR(ipUdp));
			END_IF
		END_IF				
	END_IF
END_IF
END_METHOD

{attribute 'conditionalshow'}
METHOD FB_reinit : BOOL
VAR_INPUT
END_VAR
IF (ipUdp <> 0) THEN 
	ipUdp.RegisterReceiver(localPort, THIS^);
	FB_reinit := TRUE; 
END_IF
END_METHOD

METHOD IpToLong : UDINT
VAR_INPUT
	ipAddr : T_Ipv4Addr;
END_VAR

VAR
	ipAddrArr : T_Ipv4AddrArr;
	ipAddrLong : UDINT;
END_VAR
// Scan ip string to byte array
ipAddrArr := F_ScanIPv4AddrIds(ipAddr);

// Copy bytes to ipaddrLong in reverse direction
MEMCPY(ADR(ipAddrLong) + 0, ADR(ipAddrArr) + 3, 1);
MEMCPY(ADR(ipAddrLong) + 1, ADR(ipAddrArr) + 2, 1);
MEMCPY(ADR(ipAddrLong) + 2, ADR(ipAddrArr) + 1, 1);
MEMCPY(ADR(ipAddrLong) + 3, ADR(ipAddrArr) + 0, 1); 

// Return long ip adress
IpToLong := ipAddrLong;
END_METHOD

{attribute 'object_name' := 'ReceiveData'}
{attribute 'c++_compatible'}
{attribute 'signature_flag' := '33554688'}
{attribute 'pack_mode' := '4'}
{attribute 'show'}
{attribute 'minimal_input_size' := '4'}
METHOD ReceiveData : HRESULT
VAR_INPUT
	ipAddr	: UDINT;
	udpDestPort	: UINT;
	udpSrcPort	: UINT;
	nData	: UDINT;
	pData	: PVOID;
	pVlan	: POINTER TO ETYPE_VLAN_HEADER := 0;
END_VAR
// Check data size and copy data
IF nData = nRxData THEN
	// Copy recived data
	MEMCPY(pRxData, pData, nRxData);
	
	// Increment counters
	rxCounter := rxCounter + 1;
END_IF
END_METHOD

{attribute 'object_name' := 'TcAddRef'}
{attribute 'c++_compatible'}
{attribute 'signature_flag' := '33554688'}
{attribute 'pack_mode' := '4'}
{attribute 'show'}
{attribute 'minimal_input_size' := '4'}
METHOD TcAddRef : UDINT
END_METHOD

{attribute 'object_name' := 'TcQueryInterface'}
{attribute 'c++_compatible'}
{attribute 'signature_flag' := '33554688'}
{attribute 'pack_mode' := '4'}
{attribute 'show'}
{attribute 'minimal_input_size' := '4'}
METHOD TcQueryInterface : HRESULT
VAR_INPUT
	iid	: REFERENCE TO IID;
	pipItf	: POINTER TO PVOID;
END_VAR
VAR
	ipUdpRecv : ITcIoUdpProtocolRecv;
	ipUnknown : ITcUnknown;	
END_VAR
IF GuidsEqual(ADR(iid), ADR(TC_GLOBAL_IID_LIST.IID_ITcIoUdpProtocolRecv)) THEN
	ipUdpRecv := THIS^; // cast to interface pointer
	pipItf^ := ITCUNKNOWN_TO_PVOID(ipUdpRecv);
	TcAddRef();
	TcQueryInterface := S_OK;
ELSIF GuidsEqual(ADR(iid), ADR(TC_GLOBAL_IID_LIST.IID_ITcUnknown)) THEN
	ipUnknown := THIS^; // cast to interface pointer
	pipItf^ := ITCUNKNOWN_TO_PVOID(ipUnknown);
	TcAddRef();
	TcQueryInterface := S_OK;
ELSE
	TcQueryInterface := E_HRESULTAdsErr.NOINTERFACE ; //Call super if this fb extends some other
END_IF
END_METHOD

{attribute 'object_name' := 'TcRelease'}
{attribute 'c++_compatible'}
{attribute 'signature_flag' := '33554688'}
{attribute 'pack_mode' := '4'}
{attribute 'show'}
{attribute 'minimal_input_size' := '4'}
METHOD TcRelease : UDINT
END_METHOD

END_FUNCTION_BLOCK

// ---- POUs/Interfaces/FB_StewartInterface.TcPOU
FUNCTION_BLOCK FB_StewartInterface
VAR_INPUT
	// PLC task time step
	Ts : LREAL := 0.005;
	
	// Stewart Operation 
	bStop : BOOL;
	bReset : BOOL;
	bResetScale : BOOL;
	bStart : BOOL;
	eModeCmd : E_StewartMode;
	
	// Remote data input
	bRemoteActive : BOOL := FALSE;
	uRemote : ARRAY [0..5] OF LREAL;
	uRemote_t : ARRAY [0..5] OF LREAL;
	
END_VAR
VAR_OUTPUT
	bError : BOOL;
	bBusy : BOOL := FALSE;
	bReady : BOOL := FALSE;
	eState : E_StewartState;
	eStatus : E_StewartStatus;
	eOpMode : E_StewartOpMode;
	eMode : E_StewartMode;
	
	// Feedback data
	feedback : ST_FeedbackStewart;
	
	(*
	eta : ARRAY [0..5] OF LREAL;
	eta_t : ARRAY [0..5] OF LREAL;
	eta_tt : ARRAY [0..5] OF LREAL;
	*)
	
END_VAR
VAR	
	// Hydro Simualator
	hydro : FB_HydroSimulator(0);
	
	// Stewart positon input
	u : ARRAY [0..5] OF LREAL;
	u_t : ARRAY [0..5] OF LREAL;
	uOld : ARRAY [0..5] OF LREAL;
	
	// Limted stewart setpoints
	etaRef : ARRAY [0..5] OF LREAL;
	etaRef_t : ARRAY [0..5] OF LREAL;
	etaRef_tt : ARRAY [0..5] OF LREAL;
	etaRefOld : ARRAY [0..5] OF LREAL;

	// Sine wave data
	etaSine : ARRAY [0..5] OF LREAL;
	etaSine_t : ARRAY [0..5] OF LREAL;
	etaSine_tt : ARRAY [0..5] OF LREAL;
	
	// Udp connection
	udpClient : FB_UdpClientRT('', 0, 0, 0, 0, 0, 0);	// Dummy constructor

	{attribute 'tc_no_symbol'}
	eCmnd : E_StewartCommand;
	{attribute 'tc_no_symbol'}
	rxUdp : ST_RxUdpStewart;
	{attribute 'tc_no_symbol'}
	txUdp : ST_TxUdpStewart;
	
	// Hmi connection
	txHmi : ST_TxHmiStewart;
	
	// Udp activity monitoring
	bActive : BOOL;
	frame : UDINT := 0;
	frameOld : UDINT := 0;
	frameLoss : UDINT := 0;
	
	// Time
	t : LREAL := 0.0;
	
	// Sine Generator Settings
	sineAmplitude : ARRAY [0..5] OF LREAL := [0, 0, 0.2, 2.0/180.0*PI, 2.0/180.0*PI, 0];
	sineOmega : ARRAY [0..5] OF LREAL := [0.6283, 0.6283, 0.6283, 0.6283, 0.6283, 0.6283];
	sinePhase : ARRAY [0..5] OF LREAL;

	// Zero eta
	{attribute 'tc_no_symbol'}
	etaZeros : ARRAY [0..5] OF LREAL;
	
	// Max/min settings
	etaRefMin : ARRAY [0..5] OF LREAL;
	etaRefMax : ARRAY [0..5] OF LREAL;
	
	// Soft Motion Input for Remote
	fbSoftMotion : ARRAY [0..5] OF FB_SoftMotion;
	
END_VAR

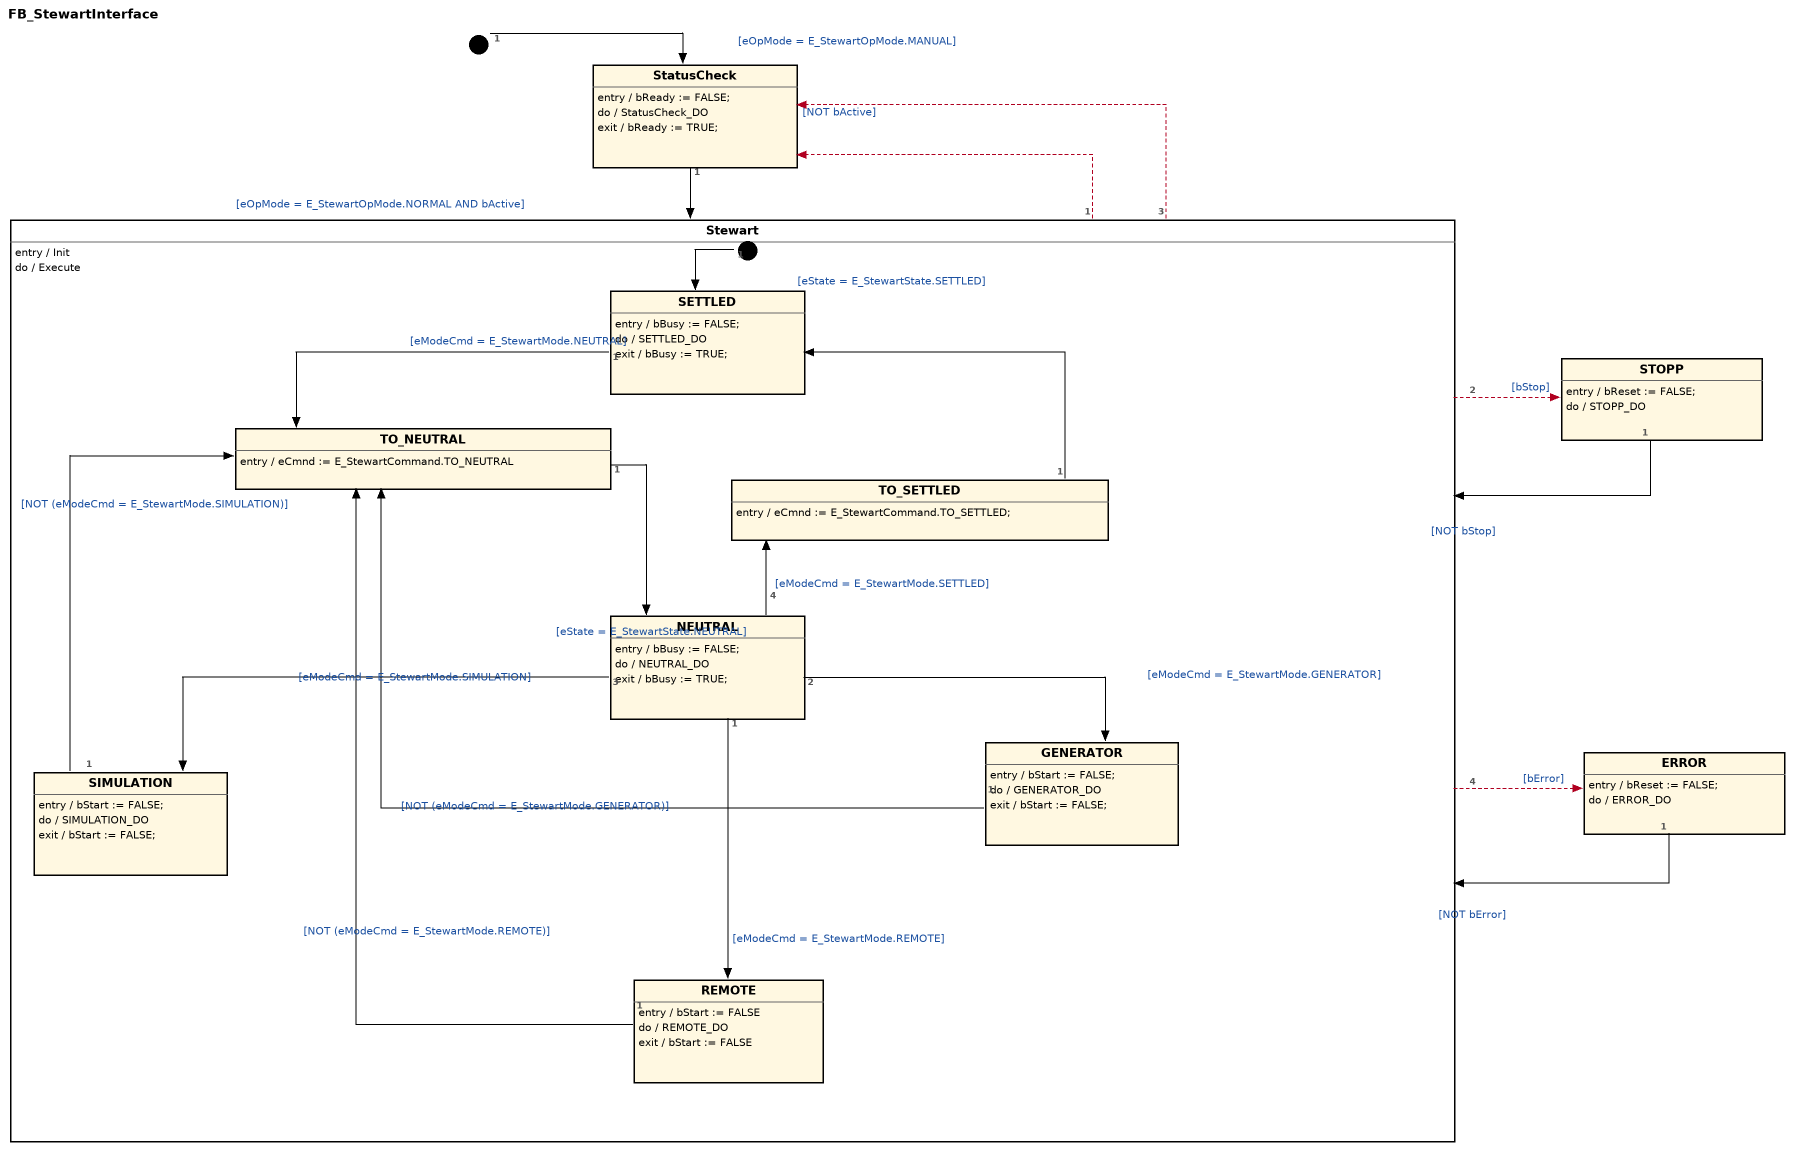
STATECHART ST_StewartInterface  // abortable
    START StartState1
    STATE StatusCheck
        entry / bReady := FALSE;
        do / StatusCheck_DO
        exit / bReady := TRUE;
    COMPOSITE STATE Stewart
        entry / Init
        do / Execute
        START StartState2
        STATE SETTLED
            entry / bBusy := FALSE;
            do / SETTLED_DO
            exit / bBusy := TRUE;
        STATE TO_NEUTRAL
            entry / eCmnd := E_StewartCommand.TO_NEUTRAL
        STATE TO_SETTLED
            entry / eCmnd := E_StewartCommand.TO_SETTLED;
        STATE NEUTRAL
            entry / bBusy := FALSE;
            do / NEUTRAL_DO
            exit / bBusy := TRUE;
        STATE GENERATOR
            entry / bStart := FALSE;
            do / GENERATOR_DO
            exit / bStart := FALSE;
        STATE SIMULATION
            entry / bStart := FALSE;
            do / SIMULATION_DO
            exit / bStart := FALSE;
        STATE REMOTE
            entry / bStart := FALSE
            do / REMOTE_DO
            exit / bStart := FALSE
        StartState2 -> SETTLED  // priority 1, on completion
        SETTLED -> TO_NEUTRAL [eModeCmd = E_StewartMode.NEUTRAL] // priority 1
        TO_NEUTRAL -> NEUTRAL [eState = E_StewartState.NEUTRAL] // priority 1
        TO_SETTLED -> SETTLED [eState = E_StewartState.SETTLED] // priority 1
        NEUTRAL -> REMOTE [eModeCmd = E_StewartMode.REMOTE] // priority 1
        NEUTRAL -> GENERATOR [eModeCmd = E_StewartMode.GENERATOR] // priority 2
        NEUTRAL -> SIMULATION [eModeCmd = E_StewartMode.SIMULATION] // priority 3
        NEUTRAL -> TO_SETTLED [eModeCmd = E_StewartMode.SETTLED] // priority 4
        GENERATOR -> TO_NEUTRAL [NOT (eModeCmd = E_StewartMode.GENERATOR)] // priority 1
        SIMULATION -> TO_NEUTRAL [NOT (eModeCmd = E_StewartMode.SIMULATION)] // priority 1
        REMOTE -> TO_NEUTRAL [NOT (eModeCmd = E_StewartMode.REMOTE)] // priority 1
    END_STATE
    STATE STOPP
        entry / bReset := FALSE;
        do / STOPP_DO
    STATE ERROR
        entry / bReset := FALSE;
        do / ERROR_DO
    StartState1 -> StatusCheck  // priority 1, on completion
    StatusCheck -> Stewart [eOpMode = E_StewartOpMode.NORMAL AND bActive] // priority 1
    Stewart -> StatusCheck [NOT bActive] // priority 1, exception
    Stewart -> STOPP [bStop] // priority 2, exception
    Stewart -> StatusCheck [eOpMode = E_StewartOpMode.MANUAL] // priority 3, exception
    Stewart -> ERROR [bError] // priority 4, exception
    STOPP -> Stewart [NOT bStop] // priority 1
    ERROR -> Stewart [NOT bError] // priority 1
END_STATECHART

METHOD decode_E_StewartOpMode : E_StewartOpMode
VAR_INPUT
	motionStatus : UDINT;
END_VAR
VAR
	mask : UDINT;
	n : USINT;
END_VAR

mask := 16#FF000000 AND motionStatus;
n := UDINT_TO_USINT(SHR(mask, 6));

(*
CASE mask OF
	16#00000000 :
		eResult := E_StewartOpMode.MANUAL;
		
	16#01000000 :
		eResult := E_StewartOpMode.NORMAL;
	
END_CASE
*)
END_METHOD

METHOD PRIVATE decode_E_StewartState : E_StewartState
VAR_INPUT
	motionStatus : UDINT;
END_VAR
VAR
	mask : UDINT;
	eResult : E_StewartState;
END_VAR
// PDF: Motion System Ethernet Interface p.18

mask := 16#0000000F AND motionStatus;

CASE mask OF
	16#00000000 : 
		eResult := E_StewartState.TRANSIT;
		
	16#00000001 : 
		eResult := E_StewartState.OFF;
		
	16#00000002 : 
		eResult := E_StewartState.SETTLED;
		
	16#00000003 : 
		eResult := E_StewartState.OIL_HEATING;
		
	16#00000004 : 
		eResult := E_StewartState.NEUTRAL;
		
	16#00000005 : 
		eResult := E_StewartState.NEUTRAL_FREEZE;
		
	16#00000008 : 
		eResult := E_StewartState.ENGAGED;
		
	16#00000009 : 
		eResult := E_StewartState.ENGAGED_FREEZE;
	
END_CASE

decode_E_StewartState := eResult;
END_METHOD

METHOD decode_E_StewartStatus : E_StewartStatus
VAR_INPUT
	motionStatus : UDINT;
END_VAR
VAR
	mask : UDINT;
	eResult : E_StewartStatus;
END_VAR

mask := 16#000000F0 AND motionStatus;

CASE mask OF
	16#00000000 :
		eResult := E_StewartStatus.SYSTEM_OK;
		
	16#01000040 :
		eResult := E_StewartStatus.WARNING;
		
	16#01000080 :
		eResult := E_StewartStatus.ERROR;
	
END_CASE

decode_E_StewartStatus := eResult;
END_METHOD

METHOD PRIVATE ERROR_DO : BOOL
VAR_INPUT
END_VAR
// Wait for SYSTEM_OK and return to settled
IF eStatus = E_StewartStatus.SYSTEM_OK THEN
	eModeCmd := E_StewartMode.SETTLED;
	eCmnd := E_StewartCommand.TO_SETTLED;

	bError := FALSE;
	
END_IF

// Check for bReset request and acknowledge fault
IF bReset THEN
	eCmnd := E_StewartCommand.ACK_FAULT;
	bReset := FALSE;
END_IF

// Execute main thread
Execute();
END_METHOD

METHOD PRIVATE Execute : BOOL
VAR_INPUT
END_VAR
VAR

	i: INT;
	
	nState : DWORD;
	nStatus : DWORD;
	nOpMode : DWORD;
	
	amp : LREAL;
	omega : LREAL;
	phi : LREAL;
	
	(*
	// Velocity boundary
	qMin : ARRAY [0..5] OF LREAL := [-0.2, -0.2, -0.2, -5.0/180.0*PI, -5.0/180.0*PI, -5.0/180.0*PI];
	qMax : ARRAY [0..5] OF LREAL := [ 0.2,  0.2,  0.2,  5.0/180.0*PI,  5.0/180.0*PI,  5.0/180.0*PI];
	V : ARRAY [0..5] OF LREAL := [6(1.0)];
	A : ARRAY [0..5] OF LREAL := [6(1.0)];
	stVelocityBoundary : ARRAY [0..5] OF ST_VelocityBoundary;
	*)
	
	
	
END_VAR
// Set etaZeros
FOR i := 0 TO 5 DO 
	etaZeros[i] := 0.0;
	
END_FOR


// Hydro Simualtor Scale reset logic
IF bResetScale THEN
	CASE eMode OF
		E_StewartMode.SETTLED, E_StewartMode.NEUTRAL :
			hydro.stInput.bReset := TRUE;
			bResetScale := FALSE;

		ELSE
			eModeCmd := E_StewartMode.NEUTRAL;				
	
	END_CASE
END_IF

// Hydro simulator
IF hydro.State = TCOM_STATE.TCOM_STATE_OP THEN
	hydro.Execute();
	hydro.stInput.bReset := FALSE;
	
END_IF

// Increment Timer
t := t + Ts;

// Set control command
txUdp.CMND := eCmnd;


(* // SOFT INPUT
// Set soft motion input
IF Ts > 0 THEN
	FOR i := 0 TO 5 DO
		// Get speed by numerical differentiation
		u_t[i] := (u[i] - uOld[i])/Ts;
		uOld[i] := u[i];
		
		fbSoftMotion[i](
			Ts := Ts,
			qRef_t := u_t[i]
		);
		
		etaRef[i] := fbSoftMotion[i].q;
		etaRef_t[i] := fbSoftMotion[i].q_t;
		
		
		
		(*
		// Apply velocity boundary
		stVelocityBoundary[i] := F_VelocityBoundary(etaRef[i], qMin[i], qMax[i], V[i], A[i], Ts);
		
		// Limit Velocity
		
		etaRef_t[i] := MAX(etaRef_t[i], stVelocityBoundary[i].qMin_t);
		etaRef_t[i] := MIN(etaRef_t[i], stVelocityBoundary[i].qMax_t);

		// Apply numerical integration based on etaRef_t
		etaRef[i] := etaRef[i] + etaRef_t[i]*Ts;

		// Absolute postion constraint
		etaRef[i] := MAX(etaRef[i], qMin[i]);
		etaRef[i] := MIN(etaRef[i], qMax[i]);
		
		// TODO: Numerical acceleration?
		*)
		
	END_FOR
	
END_IF
*)

// NO SOF STOP Motion
FOR i := 0 TO 5 DO
	etaRef[i] := LIMIT(etaRefMin[i], u[i], etaRefMax[i]);
	etaRef_t[i] := u_t[i];
 
END_FOR

// Assign motion to Stewart
txUdp.X_EXTRA 			:= LREAL_TO_REAL(etaRef[0]);
txUdp.Y_EXTRA 			:= LREAL_TO_REAL(etaRef[1]);
txUdp.Z_EXTRA 			:= LREAL_TO_REAL(etaRef[2]);
txUdp.PHI_EXTRA 		:= LREAL_TO_REAL(etaRef[3]);
txUdp.THETA_EXTRA 		:= LREAL_TO_REAL(etaRef[4]);
txUdp.PSI_EXTRA 		:= LREAL_TO_REAL(etaRef[5]);

txUdp.X_EXTRA_DOT		:= LREAL_TO_REAL(etaRef_t[0]);
txUdp.Y_EXTRA_DOT		:= LREAL_TO_REAL(etaRef_t[1]);
txUdp.Z_EXTRA_DOT		:= LREAL_TO_REAL(etaRef_t[2]);
txUdp.PHI_EXTRA_DOT		:= LREAL_TO_REAL(etaRef_t[3]);
txUdp.THETA_EXTRA_DOT	:= LREAL_TO_REAL(etaRef_t[4]);
txUdp.PSI_EXTRA_DOT		:= LREAL_TO_REAL(etaRef_t[5]);

txUdp.X_EXTRA_DDOT		:= 0.0;
txUdp.Y_EXTRA_DDOT		:= 0.0;
txUdp.Z_EXTRA_DDOT		:= 0.0;
txUdp.PHI_EXTRA_DDOT	:= 0.0;
txUdp.THETA_EXTRA_DDOT	:= 0.0;
txUdp.PSI_EXTRA_DDOT	:= 0.0;


// Update udpClient
udpClient();

// Unamsk Motion_Status signal
nState	:= 16#0000000F AND rxUdp.Motion_Status;
nStatus	:= 16#000000F0 AND rxUdp.Motion_Status;
nOpMode := 16#FF000000 AND rxUdp.Motion_Status;

// Shift for USINT conversion
nState 	:= SHR(nState, 0*4);
nStatus := SHR(nStatus, 1*4);
nOpMode := SHR(nOpMode, 6*4);

// Enum(USINT) typecast
MEMCPY(ADR(eState), ADR(nState), SIZEOF(eState));
MEMCPY(ADR(eStatus), ADR(nStatus), SIZEOF(eStatus));
MEMCPY(ADR(eOpMode), ADR(nOpMode), SIZEOF(eOpMode));

// Error/Warning check
IF (eStatus <> E_StewartStatus.SYSTEM_OK) THEN
	bError := TRUE;;
END_IF

// Check activity
frame := rxUdp.Frame_Count;
IF frame <> frameOld THEN
	// Update frame old
	frameOld := frame;
	
	// Reset frameLoss
	frameLoss := 0;
ELSE
	// Count frame losses
	frameLoss := frameLoss + 1;
END_IF

// Set activity status after 1 second given 5ms in ms
IF frameLoss > 200 THEN
	bActive := FALSE;
ELSE
	bActive := TRUE;
END_IF

// Feedback data
feedback.eta[0] := REAL_TO_LREAL(rxUdp.Actual_platform_position_surge);
feedback.eta[1] := REAL_TO_LREAL(rxUdp.Actual_platform_position_sway);
feedback.eta[2] := REAL_TO_LREAL(rxUdp.Actual_platform_position_heave);
feedback.eta[3] := REAL_TO_LREAL(rxUdp.Actual_platform_position_roll);
feedback.eta[4] := REAL_TO_LREAL(rxUdp.Actual_platform_position_pitch);
feedback.eta[5] := REAL_TO_LREAL(rxUdp.Actual_platform_position_yaw);

feedback.eta_t[0] := REAL_TO_LREAL(rxUdp.Actual_platform_velocity_surge);
feedback.eta_t[1] := REAL_TO_LREAL(rxUdp.Actual_platform_velocity_sway);
feedback.eta_t[2] := REAL_TO_LREAL(rxUdp.Actual_platform_velocity_heave);
feedback.eta_t[3] := REAL_TO_LREAL(rxUdp.Actual_platform_velocity_roll);
feedback.eta_t[4] := REAL_TO_LREAL(rxUdp.Actual_platform_velocity_pitch);
feedback.eta_t[5] := REAL_TO_LREAL(rxUdp.Actual_platform_velocity_yaw);

feedback.eta_tt[0] := REAL_TO_LREAL(rxUdp.Actual_platform_acceleration_surge);
feedback.eta_tt[1] := REAL_TO_LREAL(rxUdp.Actual_platform_acceleration_sway);
feedback.eta_tt[2] := REAL_TO_LREAL(rxUdp.Actual_platform_acceleration_heave);
feedback.eta_tt[3] := REAL_TO_LREAL(rxUdp.Actual_platform_acceleration_roll);
feedback.eta_tt[4] := REAL_TO_LREAL(rxUdp.Actual_platform_acceleration_pitch);
feedback.eta_tt[5] := REAL_TO_LREAL(rxUdp.Actual_platform_acceleration_yaw);

// Update global Hmi data
IF bActive THEN
	txHmi.status := 1;
ELSE
	txHmi.status := 0;
END_IF

txHmi.etaRef[0] := rxUdp.Platform_setpoint_surge;
txHmi.etaRef[1] := rxUdp.Platform_setpoint_sway;
txHmi.etaRef[2] := rxUdp.Platform_setpoint_heave;
txHmi.etaRef[3] := rxUdp.Platform_setpoint_roll;
txHmi.etaRef[4] := rxUdp.Platform_setpoint_pitch;
txHmi.etaRef[5] := rxUdp.Platform_setpoint_yaw;

txHmi.eta[0] := rxUdp.Actual_platform_position_surge;
txHmi.eta[1] := rxUdp.Actual_platform_position_sway;
txHmi.eta[2] := rxUdp.Actual_platform_position_heave;
txHmi.eta[3] := rxUdp.Actual_platform_position_roll;
txHmi.eta[4] := rxUdp.Actual_platform_position_pitch;
txHmi.eta[5] := rxUdp.Actual_platform_position_yaw;

txHmi.cyl[0] := rxUdp.Actual_position_actuator_1;
txHmi.cyl[1] := rxUdp.Actual_position_actuator_2;
txHmi.cyl[2] := rxUdp.Actual_position_actuator_3;
txHmi.cyl[3] := rxUdp.Actual_position_actuator_4;
txHmi.cyl[4] := rxUdp.Actual_position_actuator_5;
txHmi.cyl[5] := rxUdp.Actual_position_actuator_6;

FOR i := 0 TO 5 DO
	txHmi.dofScale[i] := LREAL_TO_REAL(hydro.stOutput.scale[i]);
END_FOR
END_METHOD

METHOD FB_exit : BOOL
VAR_INPUT
	bInCopyCode : BOOL; // if TRUE, the exit method is called for exiting an instance that is copied afterwards (online change).
END_VAR
END_METHOD

METHOD FB_init : BOOL
VAR_INPUT
	bInitRetains : BOOL; // if TRUE, the retain variables are initialized (warm start / cold start)
	bInCopyCode : BOOL;  // if TRUE, the instance afterwards gets moved into the copy code (online change)
	
	// Init variables
	_remoteIpAddr : T_Ipv4Addr;
	_remotePort : UINT;
	_localPort : UINT;
	oid : OTCID;
	

END_VAR
// Initilize udpClient
udpClient.FB_init(
	bInitRetains,
	bInCopyCode,
	_remoteIpAddr,
	_remotePort,
	_localPort,
	SIZEOF(rxUdp),
	ADR(rxUdp),
	SIZEOF(txUdp),
	ADR(txUdp)
);

// TcCOM adress
hydro.FB_init(bInitRetains, bInCopyCode, oid);

// EM8000
IF _remotePort = 50030 THEN
	rxUdp.Actual_platform_position_heave := 0.9986208;
	
	// Max/min strokes
	etaRefMin[0] := -0.2;
	etaRefMin[1] := -0.2;
	etaRefMin[2] := -0.6;
	etaRefMin[3] := -5.0/180*PI;
	etaRefMin[4] := -5.0/180*PI;
	etaRefMin[5] := -10.0/180*PI;
	
	etaRefMax[0] := 0.2;
	etaRefMax[1] := 0.2;
	etaRefMax[2] := 0.6;
	etaRefMax[3] := 5.0/180*PI;
	etaRefMax[4] := 5.0/180*PI;
	etaRefMax[5] := 10.0/180*PI;
END_IF

// EM15000
IF _remotePort = 50031 THEN
	rxUdp.Actual_platform_position_heave := 0.4663845;
	
	// Max/min strokes
	etaRefMin[0] := -0.15;
	etaRefMin[1] := -0.15;
	etaRefMin[2] := -0.3;
	etaRefMin[3] := -5.0/180*PI;
	etaRefMin[4] := -5.0/180*PI;
	etaRefMin[5] := -5.0/180*PI;
	
	etaRefMax[0] := 0.15;
	etaRefMax[1] := 0.15;
	etaRefMax[2] := 0.3;
	etaRefMax[3] := 5.0/180*PI;
	etaRefMax[4] := 5.0/180*PI;
	etaRefMax[5] := 5.0/180*PI;
END_IF
END_METHOD

METHOD FB_reinit : BOOL
VAR_INPUT
END_VAR
END_METHOD

METHOD PRIVATE GENERATOR_DO : BOOL
VAR_INPUT
END_VAR
VAR
	i : UINT;
	
	amp : LREAL;
	omega : LREAL;
	phi : LREAL;
	
END_VAR

// Apply sine generator input
FOR i := 0 TO 5 DO
	// Sine signals
	amp := sineAmplitude[i];
	omega := sineOmega[i];
	phi := sinePhase[i];
	
	u[i] := amp*SIN(omega*t + phi);
	
END_FOR


IF bStart THEN
	eCmnd := E_StewartCommand.TO_ENGAGED;
	
ELSE
	eCmnd := E_StewartCommand.TO_NEUTRAL;
	
END_IF

// Set mode
eMode := E_StewartMode.GENERATOR;
END_METHOD

METHOD PRIVATE Init
VAR_INPUT
END_VAR
// Do init here
END_METHOD

METHOD PRIVATE NEUTRAL_DO : BOOL
VAR_INPUT
END_VAR
VAR
	i : UINT;
END_VAR
// Zero input
etaRef := etaZeros;
etaRef_t := etaZeros;
etaRef_tt := etaZeros;

// Set mode
eMode := E_StewartMode.NEUTRAL;
END_METHOD

METHOD PRIVATE REMOTE_DO : BOOL
VAR_INPUT
END_VAR
VAR
	i : UINT;
	bLimitExceeded : BOOL;
	
	velocityBoundary : ARRAY [0..1] OF LREAL;
	
END_VAR

// Set input to deafult
u := uRemote;
u_t := uRemote_t;

// Enagage and disengage if remote is active
IF bStart AND bRemoteActive AND NOT bLimitExceeded THEN
	// Enagage
	eCmnd := E_StewartCommand.TO_ENGAGED;
	
ELSE
	// Resete bStart and got to Nautral
	bStart := FALSE;
	
	eCmnd := E_StewartCommand.TO_NEUTRAL;
	
END_IF


// Set mode
eMode := E_StewartMode.REMOTE;
END_METHOD

METHOD PRIVATE SETTLED_DO : BOOL
VAR_INPUT
END_VAR
VAR
	i : UINT;
END_VAR
// Zero input
etaRef := etaZeros;
etaRef_t := etaZeros;
etaRef_tt := etaZeros;


eMode := E_StewartMode.SETTLED;
END_METHOD

METHOD PRIVATE SIMULATION_DO : BOOL
VAR_INPUT
END_VAR
// Apply simulator output
u := hydro.stOutput.eta;

IF bStart THEN
	eCmnd := E_StewartCommand.TO_ENGAGED;
	
ELSE
	eCmnd := E_StewartCommand.TO_NEUTRAL;
	
END_IF
			

// Set mode
eMode := E_StewartMode.SIMULATION;
END_METHOD

METHOD PRIVATE StatusCheck_DO : BOOL
VAR_INPUT
END_VAR
eModeCmd := E_StewartMode.SETTLED;
eCmnd := E_StewartCommand.TO_SETTLED;

Execute();
END_METHOD

METHOD PRIVATE Stewart_DO : BOOL
VAR_INPUT
END_VAR

VAR
	i: INT;
END_VAR



// Execute Main thread 
Execute();
END_METHOD

METHOD PRIVATE STOPP_DO : BOOL
VAR_INPUT
END_VAR
// Got to settled in case of stop
eModeCmd := E_StewartMode.SETTLED;
eCmnd := E_StewartCommand.TO_SETTLED;
	 
// Execute main thread
Execute();

// Reset stop
IF (eStatus = E_StewartStatus.SYSTEM_OK) AND bReset THEN
	bStop := FALSE;
	
END_IF
END_METHOD

END_FUNCTION_BLOCK

// ---- HydroSimulator/FB_HydroSimulator.TcPOU
{attribute 'TcDependOnClassFactory' := 'HydroSimulator'}
FUNCTION_BLOCK FB_HydroSimulator EXTENDS FB_TcMatSimObject
VAR_INPUT
	stInput: ST_HydroSimulator_Input;
END_VAR
VAR_OUTPUT
	stOutput: ST_HydroSimulator_Output;
END_VAR
VAR
	stInitData: ST_HydroSimulatorInitData;
	arrDataAreas: ARRAY[1..2] OF ST_TcMatSimObjectDataAreaInfo;
	bParametersVerified: BOOL;
END_VAR

METHOD Execute : HRESULT

IF (SUCCEEDED(hResult)) THEN
  hResult := VerifyParameters();
END_IF

// update DataArea information
SetDataAreaInfo(ADR(arrDataAreas),2);
arrDataAreas[1].nDataAreaId := 0;
arrDataAreas[1].nSize := SIZEOF(stInput);
arrDataAreas[1].pPlcVar := ADR(stInput);
arrDataAreas[1].pModuleProcImg := 0;
arrDataAreas[1].eDataAreaType := E_TcMatSimDataAreaType.InputDst;
arrDataAreas[2].nDataAreaId := 1;
arrDataAreas[2].nSize := SIZEOF(stOutput);
arrDataAreas[2].pPlcVar := ADR(stOutput);
arrDataAreas[2].pModuleProcImg := 0;
arrDataAreas[2].eDataAreaType := E_TcMatSimDataAreaType.OutputSrc;

	
// call base method
Execute := SUPER^.Execute();
END_METHOD

METHOD FB_init : BOOL
VAR_INPUT
	/// if TRUE, the retain variables are initialized (warm start / cold start)
	bInitRetains: BOOL;
	/// if TRUE, the instance afterwards gets moved into the copy code (online change)
	bInCopyCode: BOOL;
	oid: OTCID;
END_VAR
VAR
	clsId: CLSID;
END_VAR

// initialize flags
bParametersVerified := false;
                    
// set module class id for compatibility check
clsId.Data1 := 16#1ddd7197;
clsId.Data2 := 16#7f96;
clsId.Data3 := 16#43a8;
clsId.Data4[0] := 16#9f;
clsId.Data4[1] := 16#9f;
clsId.Data4[2] := 16#ee;
clsId.Data4[3] := 16#8f;
clsId.Data4[4] := 16#6b;
clsId.Data4[5] := 16#63;
clsId.Data4[6] := 16#0d;
clsId.Data4[7] := 16#c0;

AssignClassId(clsId);
                    
// initialize InitData structure with default values              
stInitData.CallByHdr.indexGroup := 0;
stInitData.CallByHdr.indexOffset := 16#00000000;
stInitData.CallByHdr.cbData := SIZEOF(stInitData.CallBy);
stInitData.CallBy := TctModuleCallByType.CyclicTask;
stInitData.ExecutionSequenceHdr.indexGroup := 0;
stInitData.ExecutionSequenceHdr.indexOffset := 16#00000001;
stInitData.ExecutionSequenceHdr.cbData := SIZEOF(stInitData.ExecutionSequence);
stInitData.ExecutionSequence := TctModuleExecutionSequenceType.StateUpdateAfterOutputMapping;
stInitData.StepSizeHdr.indexGroup := 0;
stInitData.StepSizeHdr.indexOffset := 16#00000002;
stInitData.StepSizeHdr.cbData := SIZEOF(stInitData.StepSize);
stInitData.StepSize := TctStepSizeType.RequireMatchingTaskCycleTime;
stInitData.ExecuteModelCodeHdr.indexGroup := 0;
stInitData.ExecuteModelCodeHdr.indexOffset := 16#00000007;
stInitData.ExecuteModelCodeHdr.cbData := SIZEOF(stInitData.ExecuteModelCode);
stInitData.ExecuteModelCode := 1;
stInitData.ModelParametersHdr.indexGroup := 0;
stInitData.ModelParametersHdr.indexOffset := 16#83000000;
stInitData.ModelParametersHdr.cbData := SIZEOF(stInitData.ModelParameters);
stInitData.ModelParameters.DPController_InitialConditionFo := 0;
stInitData.ModelParameters.DetectRisePositive_vinit := 0;
stInitData.ModelParameters.Saturation_UpperSat := 1.7976931348623157e+308;
stInitData.ModelParameters.Saturation_LowerSat := 9.9999999999999995e-07;
stInitData.ModelParameters.UnitDelay_InitialCondition := 1;
stInitData.ModelParameters.Saturation1_UpperSat := 1;
stInitData.ModelParameters.Saturation1_LowerSat := 1e-10;
stInitData.ModelParameters.Integrator1_IC[0] := 0;
stInitData.ModelParameters.Integrator1_IC[1] := 0;
stInitData.ModelParameters.Integrator1_IC[2] := 0;
stInitData.ModelParameters.Integrator1_IC[3] := 0;
stInitData.ModelParameters.Integrator1_IC[4] := 0;
stInitData.ModelParameters.Integrator1_IC[5] := 0;
stInitData.ModelParameters.Integrator_IC[0] := 0;
stInitData.ModelParameters.Integrator_IC[1] := 0;
stInitData.ModelParameters.Integrator_IC[2] := 0;
stInitData.ModelParameters.Integrator_IC[3] := 0;
stInitData.ModelParameters.Integrator_IC[4] := 0;
stInitData.ModelParameters.Integrator_IC[5] := 0;
stInitData.ModelParameters.Integrator_IC_k[0] := 0;
stInitData.ModelParameters.Integrator_IC_k[1] := 0;
stInitData.ModelParameters.Integrator_IC_k[2] := 0;
stInitData.ModelParameters.Integrator_IC_k[3] := 0;
stInitData.ModelParameters.Integrator_IC_k[4] := 0;
stInitData.ModelParameters.Integrator_IC_k[5] := 0;
stInitData.ModelParameters.Integrator_IC_k[6] := 0;
stInitData.ModelParameters.Integrator_IC_k[7] := 0;
stInitData.ModelParameters.Integrator_IC_k[8] := 0;
stInitData.ModelParameters.Integrator_IC_k[9] := 0;
stInitData.ModelParameters.Integrator_IC_k[10] := 0;
stInitData.ModelParameters.Integrator_IC_k[11] := 0;
stInitData.ModelParameters.RandomSequence_Mean[0] := 0;
stInitData.ModelParameters.RandomSequence_Mean[1] := 0;
stInitData.ModelParameters.RandomSequence_Mean[2] := 0;
stInitData.ModelParameters.RandomSequence_Mean[3] := 0;
stInitData.ModelParameters.RandomSequence_Mean[4] := 0;
stInitData.ModelParameters.RandomSequence_Mean[5] := 0;
stInitData.ModelParameters.RandomSequence_StdDev[0] := 1;
stInitData.ModelParameters.RandomSequence_StdDev[1] := 1;
stInitData.ModelParameters.RandomSequence_StdDev[2] := 1;
stInitData.ModelParameters.RandomSequence_StdDev[3] := 1;
stInitData.ModelParameters.RandomSequence_StdDev[4] := 1;
stInitData.ModelParameters.RandomSequence_StdDev[5] := 1;
stInitData.ModelParameters.RandomSequence_Seed[0] := 0;
stInitData.ModelParameters.RandomSequence_Seed[1] := 20;
stInitData.ModelParameters.RandomSequence_Seed[2] := 500;
stInitData.ModelParameters.RandomSequence_Seed[3] := 9000;
stInitData.ModelParameters.RandomSequence_Seed[4] := 400;
stInitData.ModelParameters.RandomSequence_Seed[5] := 200;
stInitData.ModelParameters.Gain_Gain[0] := 10000;
stInitData.ModelParameters.Gain_Gain[1] := 10000;
stInitData.ModelParameters.Gain_Gain[2] := 100000000;
stInitData.ModelParameters.Gain_Gain[3] := 10000000;
stInitData.ModelParameters.Gain_Gain[4] := 100000000;
stInitData.ModelParameters.Gain_Gain[5] := 1000;
stInitData.ModelParameters.u_Value[0] := 0;
stInitData.ModelParameters.u_Value[1] := 0;
stInitData.ModelParameters.u_Value[2] := 0;
stInitData.ModelParameters.u_Value[3] := 0;
stInitData.ModelParameters.u_Value[4] := 0;
stInitData.ModelParameters.u_Value[5] := 0;
stInitData.ModelParameters.InputSaturation_UpperSat[0] := 0.20000000000000001;
stInitData.ModelParameters.InputSaturation_UpperSat[1] := 0.20000000000000001;
stInitData.ModelParameters.InputSaturation_UpperSat[2] := 0;
stInitData.ModelParameters.InputSaturation_UpperSat[3] := 0;
stInitData.ModelParameters.InputSaturation_UpperSat[4] := 0;
stInitData.ModelParameters.InputSaturation_UpperSat[5] := 0.087266462599716474;
stInitData.ModelParameters.InputSaturation_LowerSat[0] := -0.20000000000000001;
stInitData.ModelParameters.InputSaturation_LowerSat[1] := -0.20000000000000001;
stInitData.ModelParameters.InputSaturation_LowerSat[2] := -0;
stInitData.ModelParameters.InputSaturation_LowerSat[3] := -0;
stInitData.ModelParameters.InputSaturation_LowerSat[4] := -0;
stInitData.ModelParameters.InputSaturation_LowerSat[5] := -0.087266462599716474;
stInitData.ModelParameters.poles_Value := -30;
stInitData.ModelParameters.PolesSaturation_UpperSat := 0;
stInitData.ModelParameters.PolesSaturation_LowerSat := -30;
stInitData.ModelParameters.Constant_Value[0] := 1;
stInitData.ModelParameters.Constant_Value[1] := 1;
stInitData.ModelParameters.Constant_Value[2] := 1;
stInitData.ModelParameters.Constant_Value[3] := 1;
stInitData.ModelParameters.Constant_Value[4] := 1;
stInitData.ModelParameters.Constant_Value[5] := 1;
stInitData.ModelParameters.Constant_Value_l := 0;
stInitData.ContextInfoArr_0_TaskOidHdr.indexGroup := 0;
stInitData.ContextInfoArr_0_TaskOidHdr.indexOffset := 16#03002060;
stInitData.ContextInfoArr_0_TaskOidHdr.cbData := SIZEOF(stInitData.ContextInfoArr_0_TaskOid);
stInitData.ContextInfoArr_0_TaskPriorityHdr.indexGroup := 0;
stInitData.ContextInfoArr_0_TaskPriorityHdr.indexOffset := 16#03002070;
stInitData.ContextInfoArr_0_TaskPriorityHdr.cbData := SIZEOF(stInitData.ContextInfoArr_0_TaskPriority);
stInitData.ContextInfoArr_0_TaskCycleTimeNsHdr.indexGroup := 0;
stInitData.ContextInfoArr_0_TaskCycleTimeNsHdr.indexOffset := 16#03002080;
stInitData.ContextInfoArr_0_TaskCycleTimeNsHdr.cbData := SIZEOF(stInitData.ContextInfoArr_0_TaskCycleTimeNs);
stInitData.ContextInfoArr_0_TaskPortHdr.indexGroup := 0;
stInitData.ContextInfoArr_0_TaskPortHdr.indexOffset := 16#03002090;
stInitData.ContextInfoArr_0_TaskPortHdr.cbData := SIZEOF(stInitData.ContextInfoArr_0_TaskPort);
stInitData.ContextInfoArr_0_TaskSortOrderHdr.indexGroup := 0;
stInitData.ContextInfoArr_0_TaskSortOrderHdr.indexOffset := 16#030020b0;
stInitData.ContextInfoArr_0_TaskSortOrderHdr.cbData := SIZEOF(stInitData.ContextInfoArr_0_TaskSortOrder);
stInitData.Header.cbData := SIZEOF(stInitData)-SIZEOF(stInitData.Header);
stInitData.Header.uiElmCnt := 10;


// set pointer to InitData structure
SetInitDataInfo(ADR(stInitData));

// set DataArea information
SetDataAreaInfo(ADR(arrDataAreas),2);
arrDataAreas[1].nDataAreaId := 0;
arrDataAreas[1].nSize := SIZEOF(stInput);
arrDataAreas[1].pPlcVar := ADR(stInput);
arrDataAreas[1].pModuleProcImg := 0;
arrDataAreas[1].eDataAreaType := E_TcMatSimDataAreaType.InputDst;
arrDataAreas[2].nDataAreaId := 1;
arrDataAreas[2].nSize := SIZEOF(stOutput);
arrDataAreas[2].pPlcVar := ADR(stOutput);
arrDataAreas[2].pModuleProcImg := 0;
arrDataAreas[2].eDataAreaType := E_TcMatSimDataAreaType.OutputSrc;


// initialize basic interface pointers and return
FB_init := SUCCEEDED(Init(oid));
END_METHOD

PROPERTY InitData : ST_HydroSimulatorInitData
GET
InitData := stInitData;
END_GET
SET
stInitData := InitData;
END_SET
END_PROPERTY

{attribute 'object_name' := 'Internal_SetObjState'}
METHOD PROTECTED Internal_SetObjState
VAR_INPUT
	hr: REFERENCE TO HRESULT;
	nextState: TCOM_STATE;
END_VAR

// update pointer to InitData structure
SetInitDataInfo(ADR(stInitData));
// call base method
SUPER^.Internal_SetObjState(hr,nextState);
END_METHOD

{attribute 'object_name' := 'SaveOnlineParametersForInit'}
METHOD SaveOnlineParametersForInit : HRESULT
VAR
	idx: UINT;
	pInitElemHdr: POINTER TO TComInitDataElmHdr;
	pData: PVOID;
	nData: UDINT;
END_VAR
VAR CONSTANT
	nInitDataAlignment: UDINT := 4;
END_VAR

// update pointer to InitData structure
SetInitDataInfo(ADR(stInitData));
// call base method
SaveOnlineParametersForInit := SUPER^.SaveOnlineParametersForInit();
END_METHOD

{attribute 'object_name' := 'VerifyParameters'}
METHOD PRIVATE VerifyParameters : HRESULT
VAR
	moduleCallByParam: TctModuleCallByType;
END_VAR

IF (bParametersVerified) THEN
  VerifyParameters := Tc2_System.E_HRESULTAdsErr.HRESULT_ADS_NOERROR;
ELSE
  VerifyParameters := GetObjPara(stInitData.CallByHdr.indexOffset,SIZEOF(moduleCallByParam),ADR(moduleCallByParam));
  
  // check the "CallBy" parameter to be set to "Module"
  IF (SUCCEEDED(VerifyParameters) AND (moduleCallByParam <> TctModuleCallByType.Module)) THEN
      VerifyParameters := Tc2_System.E_HRESULTAdsErr.INVALIDPARM;
  END_IF
  
  // set the parameters verified flag
  bParametersVerified := SUCCEEDED(VerifyParameters);
END_IF
END_METHOD

END_FUNCTION_BLOCK

// ---- HydroSimulator/FB_TcMatSimObject.TcPOU
FUNCTION_BLOCK FB_TcMatSimObject
VAR_INPUT
	/// set this flag to write FB input values to the TcComObject's input DataAreas. This will overwrite the mapped input values before module execution. Set to FALSE to read the mapped input values from the TcComObject to the FB.
	bWriteFbInputValues: BOOL := TRUE;
END_VAR
VAR
	/// process image src and dst pointers and sizes
	pDataAreas: POINTER TO ST_TcMatSimObjectDataAreaInfo;
	nDataAreas: UDINT;
	/// global interface pointers
	ipObjSrv: ITComObjectServer;
	/// object interface pointers
	ipTcComObj: ITComObject;
	ipTcCyclic: ITcCyclic;
	ipTcPostCyclic: ITcPostCyclic;
	ipTcAdi: ITcADI;
	/// task interface pointers
	ipTask: ITcTask;
	/// initial parameters
	pInitData: POINTER TO TComInitDataHdr;
	/// hResult of interface calls (0 if no error)
	hResult: HRESULT;
	/// module class ID
	moduleClsId: CLSID;
	/// expected/desired module class ID
	assignedClsId: CLSID;
	bClassIdVerified: BOOL;
	/// flag indicating whether the module instance was created dynamically
	bDynInstance: BOOL;
	/// the object state at the time FB_init was called, FB_exit will try to switch to this state (only if this means to shift down)
	eInitialObjState: TCOM_STATE := TCOM_STATE.TCOM_STATE_INIT;
END_VAR

METHOD PUBLIC AssignClassId
VAR_INPUT
	clsId : CLSID;
END_VAR
assignedClsId := clsId;
bClassIdVerified := false;
END_METHOD

PROPERTY ClassId : CLSID
GET
hResult := ReadModuleClassId();
ClassId := moduleClsId;
END_GET
END_PROPERTY

PROPERTY Error : BOOL
GET
Error := FAILED(hResult);
END_GET
END_PROPERTY

PROPERTY ErrorCode : HRESULT
GET
ErrorCode := hResult;
END_GET
END_PROPERTY

{attribute 'object_name' := 'Execute'}
METHOD Execute : HRESULT
VAR
	nDaIdx: UDINT;
	pCurDataArea: POINTER TO ST_TcMatSimObjectDataAreaInfo;
END_VAR

IF (SUCCEEDED(hResult)) THEN
  hResult := VerifyClassId();
END_IF

IF (SUCCEEDED(hResult) AND State<>TCOM_STATE_OP) THEN
  hResult := Tc2_System.E_HRESULTAdsErr.NOTREADY;
END_IF

// get image pointers
IF (SUCCEEDED(hResult)) THEN
  GetImagePtrs(hResult);
END_IF

// copy inputs
IF (pDataAreas<>0 AND nDataAreas>0 AND bWriteFbInputValues) THEN
  FOR nDaIdx:=0 TO nDataAreas-1 DO
    IF (FAILED(hResult))THEN
      CONTINUE;
    END_IF
    pCurDataArea := pDataAreas + nDaIdx*SIZEOF(ST_TcMatSimObjectDataAreaInfo);
    IF ((pCurDataArea^.eDataAreaType <> E_TcMatSimDataAreaType.InputDst))THEN
      CONTINUE;
    END_IF
    IF (pCurDataArea^.pModuleProcImg<>0 AND pCurDataArea^.pPlcVar<>0) THEN
      MEMCPY(pCurDataArea^.pModuleProcImg,pCurDataArea^.pPlcVar,pCurDataArea^.nSize);
    ELSE
      hResult := Tc2_System.E_HRESULTAdsErr.NOINTERFACE;
    END_IF
  END_FOR
END_IF

// call cycle update
IF (SUCCEEDED(hResult)) THEN
  IF (ipTcCyclic<>0) THEN
    hResult := ipTcCyclic.CycleUpdate(ipTask:= ipTask, ipCaller:= 0, context:= 0);
  ELSE
    hResult := Tc2_System.E_HRESULTAdsErr.NOINTERFACE;
  END_IF
END_IF

// copy outputs
IF (pDataAreas<>0 AND nDataAreas>0) THEN
  FOR nDaIdx:=0 TO nDataAreas-1 DO
    IF (FAILED(hResult))THEN
      CONTINUE;
    END_IF
    pCurDataArea := pDataAreas + nDaIdx*SIZEOF(ST_TcMatSimObjectDataAreaInfo);
    IF ((pCurDataArea^.eDataAreaType = E_TcMatSimDataAreaType.OutputSrc) OR NOT bWriteFbInputValues) THEN
      IF (pCurDataArea^.pModuleProcImg<>0 AND pCurDataArea^.pPlcVar<>0) THEN
        MEMCPY(pCurDataArea^.pPlcVar,pCurDataArea^.pModuleProcImg,pCurDataArea^.nSize);
      ELSE
        hResult := Tc2_System.E_HRESULTAdsErr.NOINTERFACE;
      END_IF
    END_IF
  END_FOR
END_IF


// call post cyclic update
IF (SUCCEEDED(hResult)) THEN
  IF (ipTcPostCyclic<>0) THEN
    hResult := ipTcPostCyclic.PostCyclicUpdate(ipTask:= 0, ipCaller:= 0, context:= 0);
  ELSE
    hResult := Tc2_System.E_HRESULTAdsErr.NOINTERFACE;
  END_IF
END_IF

ReleaseImagePtrs();

Execute := hResult;
END_METHOD

{attribute 'object_name' := 'FB_exit'}
METHOD FB_exit : BOOL
VAR_INPUT
	/// Online Change
	bInCopyCode: BOOL;
END_VAR

IF (NOT bInCopyCode) THEN
  IF (ipObjSrv<>0) THEN
    ipObjSrv.TcRelease();
    ipObjSrv := 0;
  END_IF

  ReleaseTcComInterface();
END_IF
END_METHOD

{attribute 'object_name' := 'FB_init'}
METHOD FB_init : BOOL
VAR_INPUT
	/// init retain variables
	bInitRetains: BOOL;
	/// Online Change
	bInCopyCode: BOOL;
	oid: OTCID;
END_VAR

FB_init := SUCCEEDED(Init(oid));
END_METHOD

{attribute 'object_name' := 'GetImagePtrs'}
METHOD PRIVATE GetImagePtrs
VAR_INPUT
	hr: REFERENCE TO HRESULT;
END_VAR
VAR
	nDaIdx: UDINT;
	pCurDataArea: POINTER TO ST_TcMatSimObjectDataAreaInfo;
END_VAR

IF (ipTcAdi=0) THEN
  hr := Tc2_System.E_HRESULTAdsErr.NOINTERFACE;
END_IF
IF(State<>TCOM_STATE_OP)THEN
  hr := Tc2_System.E_HRESULTAdsErr.INVALIDSTATE;
END_IF


// get pointers to process images
IF (pDataAreas<>0 AND nDataAreas>0) THEN
  FOR nDaIdx:=0 TO nDataAreas-1 DO
    pCurDataArea := pDataAreas + nDaIdx*SIZEOF(ST_TcMatSimObjectDataAreaInfo);
    IF (FAILED(hr))THEN
      CONTINUE;
    END_IF
    IF ((pCurDataArea^.eDataAreaType <> E_TcMatSimDataAreaType.InputDst) AND (pCurDataArea^.eDataAreaType <> E_TcMatSimDataAreaType.OutputSrc))THEN
      CONTINUE;
    END_IF
    IF (pCurDataArea^.pModuleProcImg=0 AND pCurDataArea^.nSize>0) THEN
      hr := ipTcAdi.GetImagePtr(size:= pCurDataArea^.nSize , offs:=0 , adi_x:=pCurDataArea^.nDataAreaId , ppData:=ADR(pCurDataArea^.pModuleProcImg));
    END_IF
  END_FOR
END_IF

IF (FAILED(hr)) THEN
  ReleaseImagePtrs();
END_IF
END_METHOD

{attribute 'object_name' := 'GetObjPara'}
METHOD GetObjPara : HRESULT
VAR_INPUT
	pid: PTCID;
	nData: UDINT;
	pData: PVOID;
END_VAR

IF (ipTcComObj=0) THEN
  GetObjPara := Tc2_System.E_HRESULTAdsErr.NOINTERFACE;
END_IF

IF (SUCCEEDED(GetObjPara)) THEN
  GetObjPara := ipTcComObj.TcGetObjPara(pid:=pid,nData,pData,0);
END_IF
END_METHOD

{attribute 'object_name' := 'Init'}
METHOD PROTECTED Init : HRESULT
VAR_INPUT
	oid: OTCID;
END_VAR

// preinitialize variables
memset(ADR(moduleClsId),0,SIZEOF(moduleClsId));
bClassIdVerified := FALSE;
hResult := Tc2_System.E_HRESULTAdsErr.HRESULT_ADS_NOERROR;

// get object server
IF (ipObjSrv=0) THEN
  hResult := FW_ObjMgr_GetObjectServer(_AppInfo.ObjId,ADR(ipObjSrv));
END_IF

// try to get object interfaces
IF (SUCCEEDED(hresult)) THEN
  QueryTcComInterface(hResult,oid);
END_IF

// verify class id
IF (SUCCEEDED(hresult)) THEN
  hresult := VerifyClassId();
END_IF

// query interfaces, if the current state is higher than INIT
IF (SUCCEEDED(hresult) AND State>TCOM_STATE.TCOM_STATE_INIT) THEN
  QueryObjInterfaces(hResult);
END_IF

// return value
Init := hresult;
END_METHOD

{attribute 'object_name' := 'InitObjName'}
METHOD PRIVATE InitObjName
VAR_INPUT
	hr: REFERENCE TO HRESULT;
END_VAR
VAR
	objectName: STRING(255) := 'TcMatSimObject_PlcRtFbInstance';
	oid: OTCID;
END_VAR

IF (SUCCEEDED(hr)) THEN
  hr := ipTcComObj.TcGetObjectId(oid);
END_IF

IF (SUCCEEDED(hr) and bDynInstance) THEN
  objectName := TC2_STANDARD.CONCAT(objectName,'_');
  objectName := TC2_STANDARD.CONCAT(objectName,UDINT_TO_STRING(oid));
  hr := ipTcComObj.TcSetObjectName(ADR(objectName));
END_IF
END_METHOD

{attribute 'object_name' := 'Internal_SetObjState'}
METHOD PROTECTED Internal_SetObjState
VAR_INPUT
	hr: REFERENCE TO HRESULT;
	nextState: TCOM_STATE;
END_VAR

// verify class id
IF (SUCCEEDED(hr)) THEN
  hr := VerifyClassId();
END_IF

// switch object state
IF (SUCCEEDED(hr) AND nextState>=TCOM_STATE_INIT) THEN
  IF (ipTcComObj=0) THEN
    hr := Tc2_System.E_HRESULTAdsErr.NOINTERFACE;
  END_IF
  IF (ipObjSrv=0) THEN
    hr := Tc2_System.E_HRESULTAdsErr.NOINTERFACE;
  END_IF
  IF (SUCCEEDED(hr)) THEN
    hr := ipTcComObj.TcSetObjState(nextState,ipObjSrv,pInitData);
  END_IF
END_IF
END_METHOD

{attribute 'object_name' := 'QueryObjInterface'}
METHOD PRIVATE QueryObjInterface
VAR_INPUT
	hr: REFERENCE TO HRESULT;
	iid: REFERENCE TO IID;
	pipItf: POINTER TO ITcUnknown;
END_VAR
VAR CONSTANT
	pNull: PVOID := 0;
END_VAR

IF (SUCCEEDED(hr)) THEN
  IF (ipTcComObj=0) THEN
    hr := Tc2_System.E_HRESULTAdsErr.NOINTERFACE;
  ELSIF (pipItf^=ULINT_TO_DWORD(pNull)) THEN
    hr := ipTcComObj.TcQueryInterface(iid:= iid, pipItf:=pipItf);
  END_IF
END_IF
END_METHOD

{attribute 'object_name' := 'QueryObjInterfaces'}
METHOD PRIVATE QueryObjInterfaces
VAR_INPUT
	hr: REFERENCE TO HRESULT;
END_VAR

IF(State<TCOM_STATE_PREOP)THEN
  hr := Tc2_System.E_HRESULTAdsErr.INVALIDSTATE;
END_IF

//cyclic interface
QueryObjInterface(hr,IID_ITCCYCLIC,ADR(ipTcCyclic));
//post cyclic interface
QueryObjInterface(hr,IID_ITCPOSTCYCLIC,ADR(ipTcPostCyclic));
//adi interface
QueryObjInterface(hr,IID_ITcADI,ADR(ipTcAdi));
END_METHOD

{attribute 'object_name' := 'QueryTcComInterface'}
METHOD PRIVATE QueryTcComInterface
VAR_INPUT
	hr: REFERENCE TO HRESULT;
	oid: OTCID;
END_VAR

IF (ipObjSrv=0) THEN
  hr := Tc2_System.E_HRESULTAdsErr.NOINTERFACE;
END_IF

IF (SUCCEEDED(hr) AND ipTcComObj=0) THEN
  bDynInstance := FALSE;
  IF(oid>0) THEN
    // query interface of existing object
    hr := ipObjSrv.TcQueryObjectInterface(oid,IID_ITComObject,ADR(ipTcComObj));
  ELSE
    // create new instance and get the object interface
    hr := ipObjSrv.TcCreateInstance(assignedClsId,IID_ITComObject,ADR(ipTcComObj));
    IF (SUCCEEDED(hr)) THEN
      bDynInstance := TRUE;
      hr := ipTcComObj.TcSetObjectId(OTCID_CreateNewId);
    END_IF
  END_IF
  IF (SUCCEEDED(hr)) THEN
    eInitialObjState := State;
  END_IF
END_IF
END_METHOD

{attribute 'object_name' := 'ReadModuleClassId'}
METHOD PRIVATE ReadModuleClassId : HRESULT
VAR
	emptyClsId: CLSID;
END_VAR
memset(ADR(emptyClsId),0,SIZEOF(emptyClsId));
IF (memcmp(ADR(moduleClsId),ADR(emptyClsId),SIZEOF(moduleClsId))=0) THEN
  IF (ipTcComObj=0) THEN
    ReadModuleClassId := Tc2_System.E_HRESULTAdsErr.NOINTERFACE;
  END_IF

  //objectClsId := clsid;
  IF (SUCCEEDED(ReadModuleClassId)) THEN
    ReadModuleClassId := ipTcComObj.GetClassId(moduleClsId);
  END_IF
END_IF
END_METHOD

{attribute 'object_name' := 'ReleaseImagePtrs'}
METHOD PRIVATE ReleaseImagePtrs : HRESULT
VAR
	nDaIdx: UDINT;
	pCurDataArea: POINTER TO ST_TcMatSimObjectDataAreaInfo;
END_VAR

IF (ipTcAdi=0) THEN
  ReleaseImagePtrs := Tc2_System.E_HRESULTAdsErr.NOINTERFACE;
END_IF

IF (SUCCEEDED(ReleaseImagePtrs) AND pDataAreas<>0 AND nDataAreas>0) THEN
  // release pointers to the simulink module process images
  FOR nDaIdx:=0 TO nDataAreas-1 DO
    pCurDataArea := pDataAreas + nDaIdx*SIZEOF(ST_TcMatSimObjectDataAreaInfo);

    IF (pCurDataArea^.pModuleProcImg<>0) THEN
      ipTcAdi.ReleaseImagePtr(pData:=pCurDataArea^.pModuleProcImg);
      pCurDataArea^.pModuleProcImg := 0;
    END_IF
  END_FOR
END_IF
END_METHOD

{attribute 'object_name' := 'ReleaseObjInterfaces'}
METHOD PRIVATE ReleaseObjInterfaces : HRESULT

// release interface pointers
IF (ipTcCyclic<>0) THEN
  ipTcCyclic.TcRelease();
  ipTcCyclic := 0;
END_IF
IF (ipTcPostCyclic<>0) THEN
  ipTcPostCyclic.TcRelease();
  ipTcPostCyclic := 0;
END_IF
IF (ipTcAdi<>0) THEN
  ipTcAdi.TcRelease();
  ipTcAdi := 0;
END_IF
END_METHOD

{attribute 'object_name' := 'ReleaseTcComInterface'}
METHOD PRIVATE ReleaseTcComInterface : HRESULT
VAR
	nStateChangeCnt: DINT := 0;
END_VAR

IF (ipTcComObj<>0) THEN
  WHILE (State>eInitialObjState AND nStateChangeCnt<1000) DO
    State := eInitialObjState;
    nStateChangeCnt := nStateChangeCnt+1;
  END_WHILE
  ReleaseObjInterfaces();
  IF (bDynInstance) THEN
    ReleaseTcComInterface := TC3_MODULE.FW_ObjMgr_DeleteInstance(ADR(ipTcComObj));
  ELSE
    ipTcComObj.TcRelease();
  END_IF
  ipTcComObj := 0;
END_IF
END_METHOD

{attribute 'object_name' := 'ResetHresult'}
METHOD ResetHresult
hResult := S_OK;
END_METHOD

{attribute 'object_name' := 'SaveOnlineParametersForInit'}
METHOD SaveOnlineParametersForInit : HRESULT
VAR
	idx: UINT;
	pInitElemHdr: POINTER TO TComInitDataElmHdr;
	pData: PVOID;
	nData: UDINT;
END_VAR
VAR CONSTANT
	nInitDataAlignment: UDINT := 4;
END_VAR
IF (pInitData<>0) THEN
  pInitElemHdr := pInitData + SIZEOF(pInitData^);
  FOR idx:=1 TO pInitData^.uiElmCnt DO
    pData := pInitElemHdr + ULINT_TO_DWORD(SIZEOF(pInitElemHdr^));
    nData := pInitElemHdr^.cbData;
    SaveOnlineParametersForInit := GetObjPara(pInitElemHdr^.indexOffset,nData,pData);
    IF (FAILED(SaveOnlineParametersForInit)) THEN
      RETURN;
    END_IF
    pInitElemHdr := pData + (nInitDataAlignment*((nData + nInitDataAlignment - 1)/nInitDataAlignment));
  END_FOR
ELSE
	SaveOnlineParametersForInit := Tc2_System.E_HRESULTAdsErr.NOTINIT;
END_IF
END_METHOD


METHOD PUBLIC SetDataAreaInfo
VAR_INPUT
  pDataAreas: POINTER TO ST_TcMatSimObjectDataAreaInfo;
  nDataAreas: UDINT;
END_VAR

THIS^.nDataAreas := nDataAreas;
THIS^.pDataAreas := pDataAreas;
END_METHOD


METHOD PUBLIC SetInitDataInfo
VAR_INPUT
  pInitData : POINTER TO TComInitDataHdr;
END_VAR
this^.pInitData := pInitData;
END_METHOD

{attribute 'object_name' := 'SetObjPara'}
METHOD SetObjPara : HRESULT
VAR_INPUT
	pid: PTCID;
	nData: UDINT;
	pData: PVOID;
END_VAR

IF (ipTcComObj=0) THEN
  SetObjPara := Tc2_System.E_HRESULTAdsErr.NOINTERFACE;
END_IF

IF (SUCCEEDED(SetObjPara)) THEN
  SetObjPara := ipTcComObj.TcSetObjPara(pid:=pid,nData,pData,0);
END_IF
END_METHOD

{attribute 'object_name' := 'SetObjState'}
METHOD SetObjState : HRESULT
VAR_INPUT
	finalState: TCOM_STATE;
END_VAR
VAR
	bShiftUp: BOOL;
	bShiftDown: BOOL;
	currentState: TCOM_STATE;
END_VAR

currentState := State;

bShiftUp := finalState>currentState;
bShiftDown := finalState<currentState;

// do not switch up on error
IF (FAILED(hresult)) THEN
  bShiftUp := FALSE;
END_IF
// reset existing error on switching down
IF (bShiftDown) THEN
  ResetHresult();
END_IF

// prepared state switch
CASE currentState OF
  TCOM_STATE_INIT:
    IF(bShiftUp) THEN
      QueryTcComInterface(hResult,0);
      Internal_SetObjState(hResult,TCOM_STATE.TCOM_STATE_PREOP);
      InitObjName(hResult);
    END_IF

  TCOM_STATE_PREOP:
    IF(bShiftUp) THEN
      Internal_SetObjState(hResult,TCOM_STATE.TCOM_STATE_SAFEOP);
      QueryObjInterfaces(hResult);
    ELSIF (bShiftDown) THEN
      Internal_SetObjState(hResult,TCOM_STATE.TCOM_STATE_INIT);
    END_IF

  TCOM_STATE_SAFEOP:
    IF(bShiftUp) THEN
      Internal_SetObjState(hResult,TCOM_STATE.TCOM_STATE_OP);
      QueryObjInterfaces(hResult);
    ELSIF (bShiftDown) THEN
      Internal_SetObjState(hResult,TCOM_STATE.TCOM_STATE_PREOP);
      ReleaseObjInterfaces();
    END_IF


  TCOM_STATE_OP:
    IF (bShiftDown) THEN
      Internal_SetObjState(hResult,TCOM_STATE.TCOM_STATE_SAFEOP);
    END_IF
END_CASE

SetObjState := hResult;
END_METHOD

PROPERTY State : TCOM_STATE
GET
VAR
	hr: HRESULT := S_OK;
	eObjState: TCOM_STATE;
END_VAR

IF (ipTcComObj<>0) THEN
  hr := ipTcComObj.TcGetObjState(ADR(eObjState));
IF (FAILED(hr)) THEN
  eObjState := TCOM_STATE.TCOM_STATE_INIT;
END_IF
ELSE
  eObjState := TCOM_STATE.TCOM_STATE_INIT;
END_IF
State := eObjState;
END_GET
SET
SetObjState(State);
END_SET
END_PROPERTY

{attribute 'object_name' := 'VerifyClassId'}
METHOD PRIVATE VerifyClassId : HRESULT
VAR
	emptyClsId: CLSID;
END_VAR
memset(ADR(emptyClsId),0,SIZEOF(emptyClsId));
IF (bClassIdVerified) THEN
  // class ID was already verified
  VerifyClassId := Tc2_System.E_HRESULTAdsErr.HRESULT_ADS_NOERROR;
ELSIF (memcmp(ADR(assignedClsId),ADR(emptyClsId),SIZEOF(assignedClsId))=0) THEN
  // skip class ID verification if no assignedClsId specified
  VerifyClassId := Tc2_System.E_HRESULTAdsErr.HRESULT_ADS_NOERROR;
ELSE
  // verify class ID
  VerifyClassId := ReadModuleClassId();

  IF (SUCCEEDED(VerifyClassId)) THEN
    IF (memcmp(ADR(assignedClsId),ADR(moduleClsId),SIZEOF(assignedClsId))<>0) THEN
     VerifyClassId := Tc2_System.E_HRESULTAdsErr.INVALIDCLSID;
    END_IF
  END_IF
  bClassIdVerified := SUCCEEDED(VerifyClassId);
END_IF
END_METHOD

END_FUNCTION_BLOCK

// ---- POUs/Utils/FB_SoftMotion.TcPOU
FUNCTION_BLOCK FB_SoftMotion
VAR_INPUT
	Ts : LREAL := 0.01;
	qRef_t : LREAL; // Velocity reference input
	qMin : LREAL := -0.1; // Minium position
	qMax : LREAL :=  0.1; // Maximum position
	V : LREAL := 1; // Max alowable velocity
	A : LREAL := 1; // Max alowable acceleration
	
END_VAR
VAR_OUTPUT
	q : LREAL; // Limited position
	q_t : LREAL; // Limited velocity
	qMin_t : LREAL; // Current lower velocity boundary 
	qMax_t : LREAL; // Current upper velocity boundary
	
END_VAR
VAR
	t0, t1, t2 : LREAL;
	
END_VAR

// ** Velocity Boundary **
// Ensure Ts i spositive
Ts := ABS(Ts); 

// Ensure that V and A is positive
V := ABS(V);
A := ABS(A);

// Lower Boundary       
t0 := (qMin - q)/Ts;
t1 := -V;
t2 := -SQRT(ABS(2*A*(q - qMin)));
qMin_t := MAX(t0, MAX(t1, t2));

// Upper Boundary
t0 := (qMax - q)/Ts;
t1 := V;
t2 := SQRT(ABS(2*A*(qMax - q)));
qMax_t := MIN(t0, MIN(t1, t2));


// ** Calcualte Output for q and q_t **
// Limit Velocity
q_t := qRef_t;
q_t := MAX(q_t, qMin_t);
q_t := MIN(q_t, qMax_t);

// Apply numerical integration to position
q := q + q_t*Ts;

 // Ensure q is in [qMin, qMax]
q := MAX(q, qMin);
q := MIN(q, qMax);

END_FUNCTION_BLOCK

// ---- POUs/Interfaces/FB_ComauInterface.TcPOU
FUNCTION_BLOCK FB_ComauInterface
VAR_INPUT
	bStart : BOOL;
	u : ARRAY [0..5] OF LREAL;
	
END_VAR
VAR_OUTPUT
	bActive : BOOL:= FALSE;
	q : ARRAY [0..5] OF LREAL;
	q_t : ARRAY [0..5] OF LREAL;
	
END_VAR
VAR
	// Udp related
	udpClient : FB_UdpClientRT('', 0, 0, 0, 0, 0, 0);	// Dummy constructor
	
	{attribute 'tc_no_symbol'}
	rxUdp : ST_RxUdpComau;
	{attribute 'tc_no_symbol'}
	txUdp : ST_TxUdpComau;
	
	txHmi : ST_TxHmiComau;
	
	// Actviity monitoring
	frame : DINT := 0;
	frameOld : DINT := 0;
	frameLoss : DINT := 0;
	
	// Counter vsr
	i : INT;
END_VAR

// Check activity
frame := rxUdp.frameCounter;
IF frame <> frameOld THEN
	// Update frame old
	frameOld := frame;
	
	// Reset frameLoss
	frameLoss := 0;
ELSE
	// Count frame losses
	frameLoss := frameLoss + 1;
END_IF

// Set activity status after 1 second given 5ms in ms
IF frameLoss > 200 THEN
	bActive := FALSE;
ELSE
	bActive := TRUE;
END_IF

// Update udpClient
udpClient();

// Update Hmi data
UpdateHMI();

// Apply control inputs
IF bStart THEN
	txUdp.cmnd := 1;
ELSE
	txUdp.cmnd := 0;
END_IF

txUdp.udpKey := 32;

// Set contorl and feedback data
FOR i := 0 TO 5 DO
	txUdp.qDotRef[i] := LREAL_TO_REAL(u[i]);
	q[i] := rxUdp.q[i];
	q_t[i] := rxUdp.q_t[i];
	
END_FOR

METHOD FB_exit : BOOL
VAR_INPUT
	bInCopyCode : BOOL; // if TRUE, the exit method is called for exiting an instance that is copied afterwards (online change).
END_VAR
END_METHOD

METHOD FB_init : BOOL
VAR_INPUT
	bInitRetains : BOOL; // if TRUE, the retain variables are initialized (warm start / cold start)
	bInCopyCode : BOOL;  // if TRUE, the instance afterwards gets moved into the copy code (online change)
	
	// Init variables
	_remoteIpAddr : T_Ipv4Addr;
	_remotePort : UINT;
	_localPort : UINT;
END_VAR

// Initilize udpClient
udpClient.FB_init(
	bInitRetains,
	bInCopyCode,
	_remoteIpAddr,
	_remotePort,
	_localPort,
	SIZEOF(rxUdp),
	ADR(rxUdp),
	SIZEOF(txUdp),
	ADR(txUdp)
);
END_METHOD

METHOD FB_reinit : BOOL
VAR_INPUT
END_VAR
END_METHOD

METHOD UpdateHMI : BOOL
VAR_INPUT
END_VAR
VAR
	i : INT;
END_VAR
// Update HMI Data
IF bActive THEN
	txHmi.status := 1;
ELSE
	txHmi.status := 0;
END_IF

FOR i := 0 TO 5 DO
	txHmi.u[i] := LREAL_TO_REAL(u[i]);
	txHmi.q[i] := rxUdp.q[i];
	txHmi.q_t[i] := rxUdp.q_t[i];
	txHmi.qMin[i] := rxUdp.qMin[i];
	txHmi.qMax[i] := rxUdp.qMax[i];
	txHmi.qMax_t[i] := rxUdp.qMax_t[i];
END_FOR
END_METHOD

END_FUNCTION_BLOCK

// ---- POUs/Interfaces/FB_WinchInterface.TcPOU
FUNCTION_BLOCK FB_WinchInterface
VAR_INPUT
	Ts : LREAL := 0.005;
	bEnable : BOOL;
	eModeCmd : E_WinchMode;
	u : LREAL;
	uRemote : LREAL;
	
END_VAR
VAR_OUTPUT
	bActive : BOOL := FALSE;
	
	eMode : E_WinchMode;
	length : LREAL;
	length_t : LREAL;
	length_tt : LREAL;
	
	lengthUtilization : LREAL;
END_VAR
VAR
	// HMI feedback	
	pTxHmi : POINTER TO ST_TxHmiWinch;
	
	// MC2 Functions
	axis : AXIS_REF;
	fbPower : MC_Power;
	fbReset : MC_Reset;
	fbExtSetPointGenEnable : MC_ExtSetPointGenEnable;
	fbExtSetPointGenDisable : MC_ExtSetPointGenDisable;
	fbReadParameterSet : MC_ReadParameterSet;
	stAxisParameterSet : ST_AxisParameterSet;
	
	// Input trajectory
	l : LREAL := 0.0;
	l_t : LREAL := 0.0;
	l_tt : LREAL := 0.0;
	
	// Old input memeory
	uOld : LREAL;
	uRemoteOld : LREAL;
	
	// Actviity monitoring
	vel : LREAL := 0;
	velOld : LREAL := 0;
	frameLoss : DINT := 0;
	

	
END_VAR

// Read parameter set
IF NOT fbReadParameterSet.Busy AND NOT fbReadParameterSet.Error THEN
	fbReadParameterSet(
		Axis := axis,
		Parameter := stAxisParameterSet,
		Execute := TRUE
	);
	
ELSE
	fbReadParameterSet(
		Axis := axis,
		Parameter := stAxisParameterSet,
		Execute := FALSE
	);
	
END_IF

// Operation state machine
CASE eModeCmd OF
	E_WinchMode.SETTLED :
		// Reset enable
		bEnable := FALSE;
	
		// Read current state to trajectory
		l := axis.NcToPlc.ActPos;
		l_t := axis.NcToPlc.ActVelo;
		l_tt := axis.NcToPlc.ActAcc;
		
		// Disable external setpoint
		disableExtSetPoint();
		
		// Power off the drive when external setpoint is disabled
		IF NOT fbExtSetPointGenDisable.Busy AND fbExtSetPointGenDisable.Done THEN
			fbPower(
				Axis := axis,
				Enable := FALSE,
				Enable_Positive := FALSE,
				Enable_Negative := FALSE
			);
			
		END_IF
	
		// Set current mode
		eMode := eModeCmd;
		
	E_WinchMode.LOCAL, E_WinchMode.REMOTE, E_WinchMode.MOTION_COMP :		
		IF bEnable THEN
			// Enable power
			fbPower(
				Axis := axis,
				Enable := TRUE,
				Enable_Positive := TRUE,
				Enable_Negative := TRUE
			);	
			
			IF fbPower.Status THEN
				// Enable external setpoint when on
				enableExtSetPoint();
			
			END_IF
			
		ELSE
			// Disable externale setpoint
			disableExtSetPoint();
			
			IF NOT fbExtSetPointGenDisable.Busy AND fbExtSetPointGenDisable.Done THEN
				// Enable power
				fbPower(
					Axis := axis,
					Enable := FALSE,
					Enable_Positive := FALSE,
					Enable_Negative := FALSE
				);	
				
			END_IF
		END_IF
			

		IF fbPower.Status AND fbExtSetPointGenEnable.Enabled THEN			
			// Set input based on velocity input u
			CASE eMode OF
				E_WinchMode.REMOTE : 					
					l := LIMIT(stAxisParameterSet.fEncSoftEndMin, l + uRemote*Ts, stAxisParameterSet.fEncSoftEndMax);
					l_t := uRemote;
					l_tt := (uRemote - uRemoteOld)/Ts;
					
					// Update old variable
					uRemoteOld := uRemote;
					
				E_WinchMode.LOCAL, E_WinchMode.MOTION_COMP : 
					l := LIMIT(stAxisParameterSet.fEncSoftEndMin, l + u*Ts, stAxisParameterSet.fEncSoftEndMax);
					l_t := u;
					l_tt := (u - uOld)/Ts;
					
					// Update old variable
					uOld := u;
				
			END_CASE
			
			// Feed extrernal setpoints to axis interface
			MC_ExtSetPointGenFeed(
				Axis := axis,
				Position := l ,
				Velocity := l_t,
				Acceleration := l_tt,
				Direction := getDirection(l_t, l_tt)
			);
			
		END_IF
	
		// Set current mode
		eMode := eModeCmd;	
	
END_CASE

// Reset/Acknowledge errors
fbReset(
	Axis:= axis
);

// Update axis data
axis();

// Return feedback data all the time
length := axis.NcToPlc.ActPos - stAxisParameterSet.fEncSoftEndMin;
length_t := axis.NcToPlc.ActVelo;
length_tt := axis.NcToPlc.ActAcc;

// Calculate length utilization [0..100] %
IF (stAxisParameterSet.fEncSoftEndMax - stAxisParameterSet.fEncSoftEndMin) <> 0.0 THEN
	lengthUtilization := length/(stAxisParameterSet.fEncSoftEndMax - stAxisParameterSet.fEncSoftEndMin)*100;
	
ELSE
	lengthUtilization := 0;
	
END_IF

// Check activity
vel := length_t;
IF vel <> velOld THEN
	// Update frame old
	velOld := vel;
	
	// Reset frameLoss
	frameLoss := 0;
ELSE
	// Count frame losses
	frameLoss := frameLoss + 1;
END_IF

// Set activity status after 1 second given 5ms in ms
IF frameLoss > 200 THEN
	bActive := FALSE;
	
ELSE
	bActive := TRUE;
	
END_IF

METHOD PRIVATE disableExtSetPoint : BOOL
VAR_INPUT
END_VAR
fbExtSetPointGenDisable(
	Axis := axis,
	Execute := TRUE
);
fbExtSetPointGenEnable(
	Axis := axis,
	Execute := FALSE
);
END_METHOD

METHOD PRIVATE enableExtSetPoint : BOOL
VAR_INPUT
END_VAR
fbExtSetPointGenDisable(
	Axis := axis,
	Execute := FALSE
);
fbExtSetPointGenEnable(
	Axis := axis,
	Execute := TRUE
);
END_METHOD

METHOD FB_init : BOOL
VAR_INPUT
	bInitRetains : BOOL; // if TRUE, the retain variables are initialized (warm start / cold start)
	bInCopyCode : BOOL;  // if TRUE, the instance afterwards gets moved into the copy code (online change)
	
	// Init variables
	_pTxHmi : POINTER TO ST_TxHmiStewart;
END_VAR
// Ensure Power of axis is disbaled at startup
fbPower(
	Axis := axis,
	Enable := FALSE,
	Enable_Positive := FALSE,
	Enable_Negative := FALSE
);

fbExtSetPointGenDisable(
	Axis := axis,
	Execute := FALSE
);
fbExtSetPointGenEnable(
	Axis := axis,
	Execute := FALSE
);
END_METHOD

METHOD PRIVATE getDirection : DINT
VAR_INPUT
	l_t : LREAL;
	l_tt : LREAL;
END_VAR
IF l_t = 0.0 AND l_tt = 0.0 THEN
	// Standstill
	getDirection := 0;
	
ELSIF l_t >= 0.0 THEN
	// Positive motion
	getDirection := 1;
	
ELSE
	// Negative motion
	getDirection := -1;
	
END_IF
END_METHOD

METHOD PRIVATE UpdateHMI : BOOL
VAR_INPUT
END_VAR
// Update HMI variables
END_METHOD

END_FUNCTION_BLOCK

// ---- POUs/Interfaces/FB_MruInterface.TcPOU
FUNCTION_BLOCK FB_MruInterface
VAR_INPUT
END_VAR
VAR_OUTPUT
	feedback : ST_FeedbackMru;
	bActive : BOOL := FALSE;
END_VAR
VAR
	// Udp related
	udpServer : FB_UdpServerRT(0, 0, 0, 0, 0); // Dummy constructor
	
	{attribute 'tc_no_symbol'}
	rxUdpBE : ST_RxUdpMru;
	{attribute 'tc_no_symbol'}
	rxUdp : ST_RxUdpMru;
	
	// Hmi connection
	pTxHmi : POINTER TO ST_TxHmiMru;
	
	// Actviity monitoring
	frame : DINT := 0;
	frameOld : DINT := 0;
	frameLoss : DINT := 0;
END_VAR

// Check activity
frame := rxUdp.SystemTime;
IF frame <> frameOld THEN
	// Update frame old
	frameOld := frame;
	
	// Reset frameLoss
	frameLoss := 0;
ELSE
	// Count frame losses
	frameLoss := frameLoss + 1;
END_IF

// Set activity status after 1 second given 5ms in ms
IF frameLoss > 200 THEN
	bActive := FALSE;
ELSE
	bActive := TRUE;
END_IF

// Update udpServer
udpServer();

// Swap byte order on all float variables
rxUdp := BigToLittleEndian(rxUdpBE);

// ### Feedback ###
// E-Motion Body fixed positions
feedback.eta[0] := rxUdp.PosCg_F;
feedback.eta[1] := rxUdp.PosCg_S;
feedback.eta[2] := rxUdp.PosCg_D;
feedback.eta[3] := rxUdp.Roll;
feedback.eta[4] := rxUdp.Pitch;
feedback.eta[5] := rxUdp.Yaw;

// E-Motion Body fixed velocites
feedback.v[0] := rxUdp.VelCg_F;
feedback.v[1] := rxUdp.VelCg_S;
feedback.v[2] := rxUdp.VelCg_D;
feedback.v[3] := rxUdp.AngRate_R;
feedback.v[4] := rxUdp.AngRate_P;
feedback.v[5] := rxUdp.AngRate_Y;

// Update HMI Data
UpdateHMI();

METHOD BigToLittleEndian : ST_RxUdpMru 
VAR_INPUT
	rxUdpBE : ST_RxUdpMru;
END_VAR
VAR
	nData : UINT;
	n : UINT;
	pOffset : UINT;
	bytesBE : ARRAY [0..3] OF BYTE;
	bytesLE : ARRAY [0..3] OF BYTE;
	
	rxUdpLE : ST_RxUdpMru;
END_VAR
// NOTE: Only works with ST_RxMru struct!!! Not a genral function

nData := SIZEOF(rxUdpBE);

FOR n := 0 TO (nData/4 - 2) DO
	// Current pointer offset index
	pOffset := 3 + 4*n;

	IF pOffset <= nData THEN
		MEMCPY(ADR(bytesBE), ADR(rxUdpBE) + pOffset, 4);
	
		// Swap bytes from BE -> LE
		bytesLE[3] := bytesBE[0];
		bytesLE[2] := bytesBE[1];
		bytesLE[1] := bytesBE[2];
		bytesLE[0] := bytesBE[3];
		
		MEMCPY(ADR(rxUdpLE) + pOffset, ADR(bytesLE), 4);
	END_IF
END_FOR

BigToLittleEndian := rxUdpLE;
END_METHOD

METHOD FB_exit : BOOL
VAR_INPUT
	bInCopyCode : BOOL; // if TRUE, the exit method is called for exiting an instance that is copied afterwards (online change).
END_VAR
END_METHOD

METHOD FB_init : BOOL
VAR_INPUT
	bInitRetains : BOOL; // if TRUE, the retain variables are initialized (warm start / cold start)
	bInCopyCode : BOOL;  // if TRUE, the instance afterwards gets moved into the copy code (online change)
	
	// Init variables
	localPort : UINT;
	_pTxHmi : POINTER TO ST_TxHmiMru;
END_VAR
pTxHmi := _pTxHmi;

// Initilize the udpServer
udpServer.FB_init(
	bInitRetains,
	bInCopyCode,
	localPort,
	SIZEOF(rxUdpBE),
	ADR(rxUdpBE),
	0,
	0
);
END_METHOD

METHOD FB_reinit : BOOL
VAR_INPUT
END_VAR
END_METHOD

METHOD UpdateHMI
VAR_INPUT
END_VAR
VAR
	i : UINT;
END_VAR
// Update global Hmi data
IF bActive THEN
	pTxHmi^.status := 0;
ELSE
	pTxHmi^.status := -1;
END_IF

// Set MRU feedback
FOR i := 0 TO 5 DO
	pTxHmi^.eta[i] := LREAL_TO_REAL(feedback.eta[i]);
END_FOR
END_METHOD

END_FUNCTION_BLOCK

// ---- POUs/UdpFBs/FB_UdpServerRT.TcPOU
{attribute 'c++_compatible'}
FUNCTION_BLOCK FB_UdpServerRT IMPLEMENTS ITcIoUdpProtocolRecv
VAR_INPUT
	
END_VAR
VAR_OUTPUT
	rxBuffer : ARRAY [0..1023] OF BYTE;
END_VAR
VAR
	// ITcIoUdpProtocolRecv related 
	{attribute 'TcInitSymbol'}
	oid : OTCID; 
	ipUdp : ITcIoUdpProtocol;
	
	
	// Initilized variables
	localPort : UINT;
	nRxData : UDINT;
	pRxData : PVOID;
	nTxData : UDINT;
	pTxData : PVOID;
	
	// Remote specification
	remoteIpAddr : UDINT;
	remotePort : UINT;
	
	// Send/Recv counters
	rxCounter : UINT;
	txCounter : UINT;
	
	// Actual rxSize
	rxSize : UDINT;
	
	// Result
	hrInit : HRESULT;
	hrSend : HRESULT;
END_VAR

IF ipUdp <> 0 THEN
	// Check for incoming data
	ipUdp.CheckReceived();
END_IF

{attribute 'conditionalshow'}
METHOD FB_exit : BOOL
VAR_INPUT
	bInCopyCode : BOOL; // if TRUE, the exit method is called for exiting an instance that is copied afterwards (online change).
END_VAR
IF NOT bInCopyCode THEN // no online change
	IF ipUdp <> 0 THEN 
		ipUdp.UnregisterReceiver(localPort); // Shutdown
		FW_SafeRelease(ADR(ipUdp));
		FB_exit := TRUE; 
	END_IF
END_IF
END_METHOD

{attribute 'conditionalshow'}
METHOD FB_init : BOOL
VAR_INPUT
	bInitRetains : BOOL; // if TRUE, the retain variables are initialized (warm start / cold start)
	bInCopyCode : BOOL;  // if TRUE, the instance afterwards gets moved into the copy code (online change)
	
	// Init variables
	_localPort : UINT;
	_nRxData : UDINT;
	_pRxData : PVOID;
	_nTxData : UDINT;
	_pTxData : PVOID;
END_VAR
VAR
    ipSrv : ITComObjectServer;
END_VAR
// Initilize member variables
localPort := _localPort;
nRxData := _nRxData;
pRxData := _pRxData;
nTxData := _nTxData;
pTxData := _pTxData;


IF NOT bInCopyCode THEN // no online change
	IF ipUdp = 0 THEN
	    hrInit := FW_ObjMgr_GetObjectInstance(
			oid:=oid, 
			iid:=TC_GLOBAL_IID_LIST.IID_ITcIoUdpProtocol, 
			pipUnk:=ADR(ipUdp)
		);
		
		IF SUCCEEDED(hrInit) THEN 
			IF  SUCCEEDED(ipUdp.RegisterReceiver(localPort, THIS^)) THEN //open port
				FB_init := TRUE;
			ELSE 
				FW_SafeRelease(ADR(ipUdp));
			END_IF
		END_IF				
	END_IF
END_IF
END_METHOD

{attribute 'conditionalshow'}
METHOD FB_reinit : BOOL
VAR_INPUT
END_VAR
IF (ipUdp <> 0) THEN 
	ipUdp.RegisterReceiver(localPort, THIS^);
	FB_reinit := TRUE; 
END_IF
END_METHOD

{attribute 'object_name' := 'ReceiveData'}
{attribute 'c++_compatible'}
{attribute 'signature_flag' := '33554688'}
{attribute 'pack_mode' := '4'}
{attribute 'show'}
{attribute 'minimal_input_size' := '4'}
METHOD ReceiveData : HRESULT
VAR_INPUT
	ipAddr	: UDINT;
	udpDestPort	: UINT;
	udpSrcPort	: UINT;
	nData	: UDINT;
	pData	: PVOID;
	pVlan	: POINTER TO ETYPE_VLAN_HEADER := 0;
END_VAR
// Read client data
remoteIpAddr := ipAddr;
remotePort := udpSrcPort;

rxCounter := rxCounter + 1;

// Actual size fo data recevied
rxSize := nData;
MEMCPY(ADR(rxBuffer), pData, nData);

IF nData = nRxData THEN
	// Copy recived data
	MEMCPY(pRxData, pData, nRxData);
	
END_IF

IF nTxData > 0 THEN
	// Send data back to client
	hrSend := ipUdp.SendData(ipAddr, udpSrcPort, udpDestPort, nTxData, pTxData, TRUE, 0);
	txCounter := txCounter + 1;
END_IF
END_METHOD

{attribute 'object_name' := 'TcAddRef'}
{attribute 'c++_compatible'}
{attribute 'signature_flag' := '33554688'}
{attribute 'pack_mode' := '4'}
{attribute 'show'}
{attribute 'minimal_input_size' := '4'}
METHOD TcAddRef : UDINT
END_METHOD

{attribute 'object_name' := 'TcQueryInterface'}
{attribute 'c++_compatible'}
{attribute 'signature_flag' := '33554688'}
{attribute 'pack_mode' := '4'}
{attribute 'show'}
{attribute 'minimal_input_size' := '4'}
METHOD TcQueryInterface : HRESULT
VAR_INPUT
	iid	: REFERENCE TO IID;
	pipItf	: POINTER TO PVOID;
END_VAR
VAR
	ipUdpRecv : ITcIoUdpProtocolRecv;
	ipUnknown : ITcUnknown;	
END_VAR
IF GuidsEqual(ADR(iid), ADR(TC_GLOBAL_IID_LIST.IID_ITcIoUdpProtocolRecv)) THEN
	ipUdpRecv := THIS^; // cast to interface pointer
	pipItf^ := ITCUNKNOWN_TO_PVOID(ipUdpRecv);
	TcAddRef();
	TcQueryInterface := S_OK;
ELSIF GuidsEqual(ADR(iid), ADR(TC_GLOBAL_IID_LIST.IID_ITcUnknown)) THEN
	ipUnknown := THIS^; // cast to interface pointer
	pipItf^ := ITCUNKNOWN_TO_PVOID(ipUnknown);
	TcAddRef();
	TcQueryInterface := S_OK;
ELSE
	TcQueryInterface := E_HRESULTAdsErr.NOINTERFACE ; //Call super if this fb extends some other
END_IF
END_METHOD

{attribute 'object_name' := 'TcRelease'}
{attribute 'c++_compatible'}
{attribute 'signature_flag' := '33554688'}
{attribute 'pack_mode' := '4'}
{attribute 'show'}
{attribute 'minimal_input_size' := '4'}
METHOD TcRelease : UDINT
END_METHOD

END_FUNCTION_BLOCK

// ---- POUs/Interfaces/FB_QualisysInterface.TcPOU
FUNCTION_BLOCK FB_QualisysInterface
VAR_INPUT
END_VAR
VAR_OUTPUT
	bodyComponent : ST_RT6DComponent;
	markerComponent : ST_3DMarkerPositionNoLabelComponent;
	
	feedback : ST_FeedbackQualisys;
	
	bActive : BOOL := FALSE;
END_VAR
VAR
	// Udp related
	udpServer : FB_UdpServerRT(0, 0, 0, 0, 0); // Dummy constructor
	

	// Header 
	qrtPacket : ST_RTDataQRTPacket;
	qrtComponent : ARRAY [1..100] OF ST_RTComponentData;
	
	offset : UDINT;
	comp : UDINT;
	
	// HMi data
	pTxHmi : POINTER TO ST_TxHmiQualisys;
	
	// Actviity monitoring
	frame : DINT := 0;
	frameOld : DINT := 0;
	frameLoss : DINT := 0;
	
	stZero3DMarkerPositionNoLabelComponent : ST_3DMarkerPositionNoLabelComponent;
	
	// Marker tracking
	dMarker : REAL := 62.0;
	eMin : REAL;
	e : REAL;
	i : UDINT;
	j : UDINT;
	d : REAL;
	
	
	iSave : UDINT;
	jSave : UDINT;
	dSave : REAL;
	xSave : REAL;
	ySave : REAL;
	zSave : REAL;
	
	iMarker : ST_3DMarkerPositionNoLabel;
	jMarker : ST_3DMarkerPositionNoLabel;

END_VAR

// Check activity
frame := UDINT_TO_DINT(qrtPacket.nFramenumber);
IF frame <> frameOld THEN
	// Update frame old
	frameOld := frame;
	
	// Reset frameLoss
	frameLoss := 0;
ELSE
	// Count frame losses
	frameLoss := frameLoss + 1;
END_IF

// Set activity status after 1 second given 5ms in ms
IF frameLoss > 200 THEN
	bActive := FALSE;
ELSE
	bActive := TRUE;
END_IF

// Update HMI data
UpdateHMI();

// Exchange Udp data
udpServer();

// Decode Udp packet
MEMCPY(ADR(qrtPacket), ADR(udpServer.rxBuffer), SIZEOF(ST_RTDataQRTPacket));

// Zero out data
MEMCPY(ADR(markerComponent), ADR(stZero3DMarkerPositionNoLabelComponent), SIZEOF(ST_3DMarkerPositionNoLabelComponent));

offset := SIZEOF(ST_RTDataQRTPacket);
FOR comp := 1 TO qrtPacket.nComponentCount DO
	// Read components header
	MEMCPY(ADR(qrtComponent[comp]), ADR(udpServer.rxBuffer) + offset, SIZEOF(ST_RTComponentData));
	
	// Defoce components
	CASE qrtComponent[comp].nType OF
		1 : // 3D marker data 

		2 : // Unidentified 3D marker data
		MEMCPY(ADR(markerComponent), ADR(udpServer.rxBuffer) + offset, qrtComponent[comp].nSize); 
		
		3 : // Analog data from available analog devices
		
		4 : // Force data from available force plates.
		
		5 : // 6D data - position and rotation matrix
		MEMCPY(ADR(bodyComponent), ADR(udpServer.rxBuffer) + offset, qrtComponent[comp].nSize);
		
		6 : // 6D data - position and Euler angles
		
		7 : // 2D marker data
		
		8 : // Linearized 2D marker data
		
		9 : // 3D marker data with residuals
		
		10 : // Unidentified 3D marker data with residuals
		
		11 : // 6D data - position and rotation matrix with residuals
		
		12 : // 6D data - position and Euler angles with residuals
		
		13 : // Analog data from available analog devices
		
		14 : // Image frame from a specific camera
		
		15 : // Force data from available force plates
		
	END_CASE
	
